LIN {X 0,Y 162.743,Z 569.001,A -85,B 0,C 180,E1 -23228.066,E2 -23228.066} C_VEL
LIN {X 0,Y 163.505,Z 560.276,A -85,B 0,C 180,E1 -23232.409,E2 -23232.409} C_VEL
LIN {X 0,Y 164.914,Z 549.825,A -85,B 0,C 180,E1 -23236.716,E2 -23236.716} C_VEL
LIN {X 0,Y 166.509,Z 539.199,A -85,B 0,C 180,E1 -23240.376,E2 -23240.376} C_VEL
LIN {X 0,Y 168.483,Z 527.294,A -85,B 0,C 180,E1 -23243.803,E2 -23243.803} C_VEL
LIN {X 0,Y 170.774,Z 514.351,A -85,B 0,C 180,E1 -23246.914,E2 -23246.914} C_VEL
LIN {X 0,Y 173.276,Z 499.762,A -85,B 0,C 180,E1 -23249.79,E2 -23249.79} C_VEL
LIN {X 0,Y 175.692,Z 484.547,A -85,B 0,C 180,E1 -23252.203,E2 -23252.203} C_VEL
LIN {X 0,Y 177.954,Z 468.333,A -85,B 0,C 180,E1 -23254.246,E2 -23254.246} C_VEL
LIN {X 0,Y 179.877,Z 451.506,A -85,B 0,C 180,E1 -23255.876,E2 -23255.876} C_VEL
LIN {X 0,Y 183.136,Z 416.504,A -85,B 0,C 180,E1 -23258.314,E2 -23258.314} C_VEL
LIN {X 0,Y 188.818,Z 360.63,A -85,B 0,C 180,E1 -23261.887,E2 -23261.887} C_VEL
LIN {X 0,Y 177.895,Z 334.141,A -85,B 0,C 180,E1 -23265.296,E2 -23265.296} C_VEL
LIN {X 0,Y 167.703,Z 310.796,A -85,B 0,C 180,E1 -23268.793,E2 -23268.793} C_VEL
LIN {X 0,Y 164.401,Z 303.304,A -85,B 0,C 180,E1 -23270.012,E2 -23270.012} C_VEL
LIN {X 0,Y 164.284,Z 302.644,A -85,B 0,C 180,E1 -23270.145,E2 -23270.145} C_VEL
LIN {X 0,Y 164.33,Z 302.638,A -85,B 0,C 180,E1 -23274.345,E2 -23274.345} C_VEL
LIN {X 0,Y 164.369,Z 302.631,A -85,B 0,C 180,E1 -23279.127,E2 -23279.127} C_VEL
LIN {X 0,Y 164.392,Z 302.632,A -85,B 0,C 180,E1 -23284.687,E2 -23284.687} C_VEL
LIN {X 0,Y 164.435,Z 302.629,A -85,B 0,C 180,E1 -23290.092,E2 -23290.092} C_VEL
LIN {X 0,Y 164.485,Z 302.624,A -85,B 0,C 180,E1 -23295.142,E2 -23295.142} C_VEL
LIN {X 0,Y 164.797,Z 302.585,A -85,B 0,C 180,E1 -23300.175,E2 -23300.175} C_VEL
LIN {X 0,Y 164.846,Z 302.576,A -85,B 0,C 180,E1 -23302.648,E2 -23302.648} C_VEL
LIN {X 0,Y 165.043,Z 302.554,A -85,B 0,C 180,E1 -23307.556,E2 -23307.556} C_VEL
LIN {X 0,Y 165.289,Z 302.518,A -85,B 0,C 180,E1 -23309.997,E2 -23309.997} C_VEL
LIN {X 0,Y 164.765,Z 302.585,A -85,B 0,C 180,E1 -23314.89,E2 -23314.89} C_VEL
LIN {X 0,Y 164.847,Z 302.577,A -85,B 0,C 180,E1 -23317.345,E2 -23317.345} C_VEL
LIN {X 0,Y 164.735,Z 302.585,A -85,B 0,C 180,E1 -23321.129,E2 -23321.129} C_VEL
LIN {X 0,Y 164.475,Z 302.619,A -85,B 0,C 180,E1 -23327.4,E2 -23327.4} C_VEL
LIN {X 0,Y 164.464,Z 302.621,A -85,B 0,C 180,E1 -23329.987,E2 -23329.987} C_VEL
LIN {X 0,Y 164.383,Z 302.629,A -85,B 0,C 180,E1 -23336.131,E2 -23336.131} C_VEL
LIN {X 0,Y 164.363,Z 302.637,A -85,B 0,C 180,E1 -23341.225,E2 -23341.225} C_VEL
LIN {X 0,Y 164.3,Z 302.64,A -85,B 0,C 180,E1 -23346.783,E2 -23346.783} C_VEL
LIN {X 0,Y 164.288,Z 302.645,A -85,B 0,C 180,E1 -23349.912,E2 -23349.912} C_VEL
LIN {X 0,Y 164.267,Z 302.644,A -85,B 0,C 180,E1 -23353.341,E2 -23353.341} C_VEL
LIN {X 0,Y 164.251,Z 302.649,A -85,B 0,C 180,E1 -23356.798,E2 -23356.798} C_VEL
LIN {X 0,Y 164.283,Z 302.644,A -85,B 0,C 180,E1 -23360.351,E2 -23360.351} C_VEL
LIN {X 0,Y 164.317,Z 302.641,A -85,B 0,C 180,E1 -23366.222,E2 -23366.222} C_VEL
LIN {X 0,Y 164.393,Z 302.63,A -85,B 0,C 180,E1 -23369.138,E2 -23369.138} C_VEL
LIN {X 0,Y 164.394,Z 302.632,A -85,B 0,C 180,E1 -23374.693,E2 -23374.693} C_VEL
LIN {X 0,Y 164.472,Z 302.618,A -85,B 0,C 180,E1 -23380.052,E2 -23380.052} C_VEL
LIN {X 0,Y 164.524,Z 302.616,A -85,B 0,C 180,E1 -23385.151,E2 -23385.151} C_VEL
LIN {X 0,Y 164.797,Z 302.58,A -85,B 0,C 180,E1 -23390.18,E2 -23390.18} C_VEL
LIN {X 0,Y 164.839,Z 302.577,A -85,B 0,C 180,E1 -23392.653,E2 -23392.653} C_VEL
LIN {X 0,Y 165.038,Z 302.551,A -85,B 0,C 180,E1 -23397.561,E2 -23397.561} C_VEL
LIN {X 0,Y 165.285,Z 302.52,A -85,B 0,C 180,E1 -23400.002,E2 -23400.002} C_VEL
LIN {X 0,Y 164.76,Z 302.587,A -85,B 0,C 180,E1 -23404.896,E2 -23404.896} C_VEL
LIN {X 0,Y 164.841,Z 302.576,A -85,B 0,C 180,E1 -23407.35,E2 -23407.35} C_VEL
LIN {X 0,Y 164.745,Z 302.59,A -85,B 0,C 180,E1 -23411.154,E2 -23411.154} C_VEL
LIN {X 0,Y 164.476,Z 302.624,A -85,B 0,C 180,E1 -23417.406,E2 -23417.406} C_VEL
LIN {X 0,Y 164.465,Z 302.626,A -85,B 0,C 180,E1 -23419.992,E2 -23419.992} C_VEL
LIN {X 0,Y 164.379,Z 302.637,A -85,B 0,C 180,E1 -23426.131,E2 -23426.131} C_VEL
LIN {X 0,Y 164.382,Z 302.636,A -85,B 0,C 180,E1 -23431.239,E2 -23431.239} C_VEL
LIN {X 0,Y 164.351,Z 302.637,A -85,B 0,C 180,E1 -23437.545,E2 -23437.545} C_VEL
LIN {X 0,Y 164.407,Z 302.858,A -85,B 0,C 180,E1 -23438.014,E2 -23438.014} C_VEL
LIN {X 0,Y 174.424,Z 329.86,A -85,B 0,C 180,E1 -23441.961,E2 -23441.961} C_VEL
LIN {X 0,Y 184.34,Z 358.027,A -85,B 0,C 180,E1 -23445.535,E2 -23445.535} C_VEL
LIN {X 0,Y 188.983,Z 371.855,A -85,B 0,C 180,E1 -23447.122,E2 -23447.122} C_VEL
LIN {X 0,Y 189.295,Z 378.263,A -85,B 0,C 180,E1 -23447.63,E2 -23447.63} C_VEL
LIN {X 0,Y 180.179,Z 471.457,A -85,B 0,C 180,E1 -23453.85,E2 -23453.85} C_VEL
LIN {X 0,Y 178.064,Z 488.079,A -85,B 0,C 180,E1 -23455.437,E2 -23455.437} C_VEL
LIN {X 0,Y 175.518,Z 504.903,A -85,B 0,C 180,E1 -23457.572,E2 -23457.572} C_VEL
LIN {X 0,Y 172.894,Z 520.655,A -85,B 0,C 180,E1 -23460.139,E2 -23460.139} C_VEL
LIN {X 0,Y 170.429,Z 534.802,A -85,B 0,C 180,E1 -23463.029,E2 -23463.029} C_VEL
LIN {X 0,Y 168.143,Z 547.791,A -85,B 0,C 180,E1 -23466.283,E2 -23466.283} C_VEL
LIN {X 0,Y 167.894,Z 549.217,A -85,B 0,C 180,E1 -23466.688,E2 -23466.688} C_VEL
LIN {X 0,Y 166.516,Z 553.567,A -85,B 0,C 180,E1 -23467.983,E2 -23467.983} C_VEL
LIN {X 0,Y 162.593,Z 560.027,A -85,B 0,C 180,E1 -23470.217,E2 -23470.217} C_VEL
LIN {X 0,Y 158.866,Z 566.141,A -85,B 0,C 180,E1 -23472.686,E2 -23472.686} C_VEL
LIN {X 0,Y 157.82,Z 569.902,A -85,B 0,C 180,E1 -23474.303,E2 -23474.303} C_VEL
LIN {X 0,Y 157.069,Z 578.706,A -85,B 0,C 180,E1 -23478.388,E2 -23478.388} C_VEL
LIN {X 0,Y 156.845,Z 586.764,A -85,B 0,C 180,E1 -23482.925,E2 -23482.925} C_VEL
LIN {X 0,Y 156.901,Z 591.497,A -85,B 0,C 180,E1 -23486.151,E2 -23486.151} C_VEL
LIN {X 0,Y 156.999,Z 596.192,A -85,B 0,C 180,E1 -23490.004,E2 -23490.004} C_VEL
LIN {X 0,Y 156.404,Z 599.726,A -85,B 0,C 180,E1 -23493.868,E2 -23493.868} C_VEL
LIN {X 0,Y 156.018,Z 602.437,A -85,B 0,C 180,E1 -23497.77,E2 -23497.77} C_VEL
LIN {X 0,Y 156.148,Z 605.076,A -85,B 0,C 180,E1 -23503.009,E2 -23503.009} C_VEL
LIN {X 0,Y 157.589,Z 606.716,A -85,B 0,C 180,E1 -23508.194,E2 -23508.194} C_VEL
LIN {X 0,Y 160.486,Z 607.537,A -85,B 0,C 180,E1 -23513.215,E2 -23513.215} C_VEL
LIN {X 0,Y 167.481,Z 607.223,A -85,B 0,C 180,E1 -23520.239,E2 -23520.239} C_VEL
LIN {X 0,Y 177.074,Z 605.132,A -85,B 0,C 180,E1 -23526.541,E2 -23526.541} C_VEL
LIN {X 0,Y 185.072,Z 602.786,A -85,B 0,C 180,E1 -23530.211,E2 -23530.211} C_VEL
LIN {X 0,Y 194.013,Z 599.774,A -85,B 0,C 180,E1 -23533.496,E2 -23533.496} C_VEL
LIN {X 0,Y 205.058,Z 595.453,A -85,B 0,C 180,E1 -23536.726,E2 -23536.726} C_VEL
LIN {X 0,Y 205.719,Z 595.098,A -85,B 0,C 180,E1 -23537.233,E2 -23537.233} C_VEL
LIN {X 0,Y 196.732,Z 597.398,A -85,B 0,C 180,E1 -23539.98,E2 -23539.98} C_VEL
LIN {X 0,Y 183.81,Z 599.568,A -85,B 0,C 180,E1 -23545.002,E2 -23545.002} C_VEL
LIN {X 0,Y 176.253,Z 599.98,A -85,B 0,C 180,E1 -23548.775,E2 -23548.775} C_VEL
LIN {X 0,Y 169.945,Z 599.539,A -85,B 0,C 180,E1 -23552.94,E2 -23552.94} C_VEL
LIN {X 0,Y 164.67,Z 598.231,A -85,B 0,C 180,E1 -23557.409,E2 -23557.409} C_VEL
LIN {X 0,Y 160.779,Z 596.017,A -85,B 0,C 180,E1 -23562.181,E2 -23562.181} C_VEL
LIN {X 0,Y 157.895,Z 592.902,A -85,B 0,C 180,E1 -23567.139,E2 -23567.139} C_VEL
LIN {X 0,Y 155.901,Z 587.493,A -85,B 0,C 180,E1 -23573.533,E2 -23573.533} C_VEL
LIN {X 0,Y 155.54,Z 583.386,A -85,B 0,C 180,E1 -23577.408,E2 -23577.408} C_VEL
LIN {X 0,Y 155.366,Z 578.521,A -85,B 0,C 180,E1 -23581.294,E2 -23581.294} C_VEL
LIN {X 0,Y 155.54,Z 571.047,A -85,B 0,C 180,E1 -23586.222,E2 -23586.222} C_VEL
LIN {X 0,Y 156.083,Z 563.476,A -85,B 0,C 180,E1 -23590.374,E2 -23590.374} C_VEL
LIN {X 0,Y 157.215,Z 553.624,A -85,B 0,C 180,E1 -23594.892,E2 -23594.892} C_VEL
LIN {X 0,Y 158.614,Z 543.638,A -85,B 0,C 180,E1 -23598.736,E2 -23598.736} C_VEL
LIN {X 0,Y 160.777,Z 530.826,A -85,B 0,C 180,E1 -23602.825,E2 -23602.825} C_VEL
LIN {X 0,Y 163.25,Z 516.685,A -85,B 0,C 180,E1 -23606.527,E2 -23606.527} C_VEL
LIN {X 0,Y 165.685,Z 502.525,A -85,B 0,C 180,E1 -23609.543,E2 -23609.543} C_VEL
LIN {X 0,Y 168.246,Z 487.239,A -85,B 0,C 180,E1 -23612.178,E2 -23612.178} C_VEL
LIN {X 0,Y 170.757,Z 470.23,A -85,B 0,C 180,E1 -23614.477,E2 -23614.477} C_VEL
LIN {X 0,Y 172.789,Z 453.3,A -85,B 0,C 180,E1 -23616.228,E2 -23616.228} C_VEL
LIN {X 0,Y 175.716,Z 422.77,A -85,B 0,C 180,E1 -23618.492,E2 -23618.492} C_VEL
LIN {X 0,Y 181.978,Z 362.013,A -85,B 0,C 180,E1 -23622.588,E2 -23622.588} C_VEL
LIN {X 0,Y 171.144,Z 335.711,A -85,B 0,C 180,E1 -23626.13,E2 -23626.13} C_VEL
LIN {X 0,Y 160.884,Z 312.149,A -85,B 0,C 180,E1 -23629.833,E2 -23629.833} C_VEL
LIN {X 0,Y 157.365,Z 304.37,A -85,B 0,C 180,E1 -23631.187,E2 -23631.187} C_VEL
LIN {X 0,Y 157.203,Z 303.526,A -85,B 0,C 180,E1 -23631.408,E2 -23631.408} C_VEL
LIN {X 0,Y 157.278,Z 303.516,A -85,B 0,C 180,E1 -23634.482,E2 -23634.482} C_VEL
LIN {X 0,Y 157.282,Z 303.516,A -85,B 0,C 180,E1 -23638.098,E2 -23638.098} C_VEL
LIN {X 0,Y 157.307,Z 303.515,A -85,B 0,C 180,E1 -23643.46,E2 -23643.46} C_VEL
LIN {X 0,Y 157.374,Z 303.511,A -85,B 0,C 180,E1 -23649.681,E2 -23649.681} C_VEL
LIN {X 0,Y 157.419,Z 303.504,A -85,B 0,C 180,E1 -23654.459,E2 -23654.459} C_VEL
LIN {X 0,Y 157.722,Z 303.468,A -85,B 0,C 180,E1 -23659.729,E2 -23659.729} C_VEL
LIN {X 0,Y 157.803,Z 303.453,A -85,B 0,C 180,E1 -23662.318,E2 -23662.318} C_VEL
LIN {X 0,Y 158.251,Z 303.395,A -85,B 0,C 180,E1 -23669.997,E2 -23669.997} C_VEL
LIN {X 0,Y 157.803,Z 303.452,A -85,B 0,C 180,E1 -23677.675,E2 -23677.675} C_VEL
LIN {X 0,Y 157.665,Z 303.466,A -85,B 0,C 180,E1 -23681.299,E2 -23681.299} C_VEL
LIN {X 0,Y 157.446,Z 303.498,A -85,B 0,C 180,E1 -23685.531,E2 -23685.531} C_VEL
LIN {X 0,Y 157.361,Z 303.506,A -85,B 0,C 180,E1 -23690.93,E2 -23690.93} C_VEL
LIN {X 0,Y 157.304,Z 303.51,A -85,B 0,C 180,E1 -23696.682,E2 -23696.682} C_VEL
LIN {X 0,Y 157.265,Z 303.519,A -85,B 0,C 180,E1 -23702.425,E2 -23702.425} C_VEL
LIN {X 0,Y 157.269,Z 303.515,A -85,B 0,C 180,E1 -23706.454,E2 -23706.454} C_VEL
LIN {X 0,Y 157.201,Z 303.525,A -85,B 0,C 180,E1 -23712.109,E2 -23712.109} C_VEL
LIN {X 0,Y 157.181,Z 303.53,A -85,B 0,C 180,E1 -23717.883,E2 -23717.883} C_VEL
LIN {X 0,Y 157.255,Z 303.519,A -85,B 0,C 180,E1 -23723.55,E2 -23723.55} C_VEL
LIN {X 0,Y 157.289,Z 303.515,A -85,B 0,C 180,E1 -23728.091,E2 -23728.091} C_VEL
LIN {X 0,Y 157.303,Z 303.516,A -85,B 0,C 180,E1 -23733.465,E2 -23733.465} C_VEL
LIN {X 0,Y 157.38,Z 303.502,A -85,B 0,C 180,E1 -23739.67,E2 -23739.67} C_VEL
LIN {X 0,Y 157.45,Z 303.496,A -85,B 0,C 180,E1 -23744.468,E2 -23744.468} C_VEL
LIN {X 0,Y 157.723,Z 303.461,A -85,B 0,C 180,E1 -23749.735,E2 -23749.735} C_VEL
LIN {X 0,Y 157.797,Z 303.453,A -85,B 0,C 180,E1 -23752.324,E2 -23752.324} C_VEL
LIN {X 0,Y 158.247,Z 303.396,A -85,B 0,C 180,E1 -23760.002,E2 -23760.002} C_VEL
LIN {X 0,Y 157.799,Z 303.453,A -85,B 0,C 180,E1 -23767.68,E2 -23767.68} C_VEL
LIN {X 0,Y 157.673,Z 303.47,A -85,B 0,C 180,E1 -23771.322,E2 -23771.322} C_VEL
LIN {X 0,Y 157.453,Z 303.498,A -85,B 0,C 180,E1 -23775.536,E2 -23775.536} C_VEL
LIN {X 0,Y 157.359,Z 303.513,A -85,B 0,C 180,E1 -23780.936,E2 -23780.936} C_VEL
LIN {X 0,Y 157.302,Z 303.52,A -85,B 0,C 180,E1 -23786.684,E2 -23786.684} C_VEL
LIN {X 0,Y 157.275,Z 303.521,A -85,B 0,C 180,E1 -23792.43,E2 -23792.43} C_VEL
LIN {X 0,Y 157.299,Z 303.662,A -85,B 0,C 180,E1 -23796.782,E2 -23796.782} C_VEL
LIN {X 0,Y 158.315,Z 306.417,A -85,B 0,C 180,E1 -23797.23,E2 -23797.23} C_VEL
LIN {X 0,Y 161.302,Z 313.749,A -85,B 0,C 180,E1 -23798.451,E2 -23798.451} C_VEL
LIN {X 0,Y 170.717,Z 339.571,A -85,B 0,C 180,E1 -23802.219,E2 -23802.219} C_VEL
LIN {X 0,Y 181.836,Z 371.924,A -85,B 0,C 180,E1 -23806.307,E2 -23806.307} C_VEL
LIN {X 0,Y 182.488,Z 374.64,A -85,B 0,C 180,E1 -23806.593,E2 -23806.593} C_VEL
LIN {X 0,Y 182.512,Z 379.17,A -85,B 0,C 180,E1 -23806.945,E2 -23806.945} C_VEL
LIN {X 0,Y 173.291,Z 470.889,A -85,B 0,C 180,E1 -23813.354,E2 -23813.354} C_VEL
LIN {X 0,Y 171.029,Z 488.174,A -85,B 0,C 180,E1 -23815.09,E2 -23815.09} C_VEL
LIN {X 0,Y 168.568,Z 504.001,A -85,B 0,C 180,E1 -23817.184,E2 -23817.184} C_VEL
LIN {X 0,Y 165.952,Z 519.55,A -85,B 0,C 180,E1 -23819.812,E2 -23819.812} C_VEL
LIN {X 0,Y 163.44,Z 533.752,A -85,B 0,C 180,E1 -23822.818,E2 -23822.818} C_VEL
LIN {X 0,Y 160.98,Z 547.649,A -85,B 0,C 180,E1 -23826.468,E2 -23826.468} C_VEL
LIN {X 0,Y 159.258,Z 558.77,A -85,B 0,C 180,E1 -23830.005,E2 -23830.005} C_VEL
LIN {X 0,Y 157.82,Z 569.902,A -85,B 0,C 180,E1 -23834.303,E2 -23834.303} C_VEL
LIN {X 0,Y 156.843,Z 573.57,A -85,B 0,C 180,E1 -23835.974,E2 -23835.974} C_VEL
LIN {X 0,Y 153.579,Z 578.678,A -85,B 0,C 180,E1 -23838.872,E2 -23838.872} C_VEL
LIN {X 0,Y 150.589,Z 583.4,A -85,B 0,C 180,E1 -23841.995,E2 -23841.995} C_VEL
LIN {X 0,Y 150.048,Z 586.324,A -85,B 0,C 180,E1 -23843.952,E2 -23843.952} C_VEL
LIN {X 0,Y 150.095,Z 592.612,A -85,B 0,C 180,E1 -23848.662,E2 -23848.662} C_VEL
LIN {X 0,Y 150.058,Z 595.5,A -85,B 0,C 180,E1 -23851.346,E2 -23851.346} C_VEL
LIN {X 0,Y 149.38,Z 598.925,A -85,B 0,C 180,E1 -23855.403,E2 -23855.403} C_VEL
LIN {X 0,Y 149.055,Z 602.289,A -85,B 0,C 180,E1 -23860.875,E2 -23860.875} C_VEL
LIN {X 0,Y 149.939,Z 604.692,A -85,B 0,C 180,E1 -23866.337,E2 -23866.337} C_VEL
LIN {X 0,Y 153.688,Z 606.534,A -85,B 0,C 180,E1 -23873.85,E2 -23873.85} C_VEL
LIN {X 0,Y 158.571,Z 606.846,A -85,B 0,C 180,E1 -23879.182,E2 -23879.182} C_VEL
LIN {X 0,Y 164.389,Z 606.36,A -85,B 0,C 180,E1 -23883.768,E2 -23883.768} C_VEL
LIN {X 0,Y 171.405,Z 605.089,A -85,B 0,C 180,E1 -23887.958,E2 -23887.958} C_VEL
LIN {X 0,Y 179.732,Z 603.155,A -85,B 0,C 180,E1 -23891.666,E2 -23891.666} C_VEL
LIN {X 0,Y 188.963,Z 600.49,A -85,B 0,C 180,E1 -23894.967,E2 -23894.967} C_VEL
LIN {X 0,Y 196.373,Z 598.06,A -85,B 0,C 180,E1 -23897.155,E2 -23897.155} C_VEL
LIN {X 0,Y 186.819,Z 599.715,A -85,B 0,C 180,E1 -23900.242,E2 -23900.242} C_VEL
LIN {X 0,Y 178.099,Z 600.588,A -85,B 0,C 180,E1 -23903.705,E2 -23903.705} C_VEL
LIN {X 0,Y 170.245,Z 600.644,A -85,B 0,C 180,E1 -23907.542,E2 -23907.542} C_VEL
LIN {X 0,Y 163.653,Z 599.866,A -85,B 0,C 180,E1 -23911.809,E2 -23911.809} C_VEL
LIN {X 0,Y 158.138,Z 598.221,A -85,B 0,C 180,E1 -23916.421,E2 -23916.421} C_VEL
LIN {X 0,Y 154.048,Z 595.742,A -85,B 0,C 180,E1 -23921.374,E2 -23921.374} C_VEL
LIN {X 0,Y 150.434,Z 591.275,A -85,B 0,C 180,E1 -23927.862,E2 -23927.862} C_VEL
LIN {X 0,Y 148.924,Z 586.344,A -85,B 0,C 180,E1 -23933.393,E2 -23933.393} C_VEL
LIN {X 0,Y 148.548,Z 582.223,A -85,B 0,C 180,E1 -23937.286,E2 -23937.286} C_VEL
LIN {X 0,Y 148.356,Z 577.075,A -85,B 0,C 180,E1 -23941.355,E2 -23941.355} C_VEL
LIN {X 0,Y 148.596,Z 569.035,A -85,B 0,C 180,E1 -23946.652,E2 -23946.652} C_VEL
LIN {X 0,Y 149.305,Z 559.986,A -85,B 0,C 180,E1 -23951.538,E2 -23951.538} C_VEL
LIN {X 0,Y 150.691,Z 549.471,A -85,B 0,C 180,E1 -23956.248,E2 -23956.248} C_VEL
LIN {X 0,Y 152.242,Z 538.695,A -85,B 0,C 180,E1 -23960.254,E2 -23960.254} C_VEL
LIN {X 0,Y 154.419,Z 526.049,A -85,B 0,C 180,E1 -23964.178,E2 -23964.178} C_VEL
LIN {X 0,Y 156.905,Z 512.255,A -85,B 0,C 180,E1 -23967.689,E2 -23967.689} C_VEL
LIN {X 0,Y 159.536,Z 497.226,A -85,B 0,C 180,E1 -23970.802,E2 -23970.802} C_VEL
LIN {X 0,Y 162.227,Z 480.769,A -85,B 0,C 180,E1 -23973.526,E2 -23973.526} C_VEL
LIN {X 0,Y 164.6,Z 463.974,A -85,B 0,C 180,E1 -23975.659,E2 -23975.659} C_VEL
LIN {X 0,Y 166.526,Z 446.338,A -85,B 0,C 180,E1 -23977.347,E2 -23977.347} C_VEL
LIN {X 0,Y 175.189,Z 363.631,A -85,B 0,C 180,E1 -23983.28,E2 -23983.28} C_VEL
LIN {X 0,Y 164.621,Z 337.772,A -85,B 0,C 180,E1 -23986.912,E2 -23986.912} C_VEL
LIN {X 0,Y 153.612,Z 312.55,A -85,B 0,C 180,E1 -23991.099,E2 -23991.099} C_VEL
LIN {X 0,Y 150.299,Z 305.128,A -85,B 0,C 180,E1 -23992.454,E2 -23992.454} C_VEL
LIN {X 0,Y 150.197,Z 304.402,A -85,B 0,C 180,E1 -23992.639,E2 -23992.639} C_VEL
LIN {X 0,Y 150.208,Z 304.402,A -85,B 0,C 180,E1 -23997.368,E2 -23997.368} C_VEL
LIN {X 0,Y 150.237,Z 304.395,A -85,B 0,C 180,E1 -24002.718,E2 -24002.718} C_VEL
LIN {X 0,Y 150.336,Z 304.386,A -85,B 0,C 180,E1 -24009.216,E2 -24009.216} C_VEL
LIN {X 0,Y 150.327,Z 304.389,A -85,B 0,C 180,E1 -24013.706,E2 -24013.706} C_VEL
LIN {X 0,Y 150.643,Z 304.347,A -85,B 0,C 180,E1 -24019.241,E2 -24019.241} C_VEL
LIN {X 0,Y 150.737,Z 304.335,A -85,B 0,C 180,E1 -24021.956,E2 -24021.956} C_VEL
LIN {X 0,Y 151.212,Z 304.272,A -85,B 0,C 180,E1 -24029.996,E2 -24029.996} C_VEL
LIN {X 0,Y 150.737,Z 304.331,A -85,B 0,C 180,E1 -24038.037,E2 -24038.037} C_VEL
LIN {X 0,Y 150.599,Z 304.347,A -85,B 0,C 180,E1 -24041.489,E2 -24041.489} C_VEL
LIN {X 0,Y 150.353,Z 304.379,A -85,B 0,C 180,E1 -24046.284,E2 -24046.284} C_VEL
LIN {X 0,Y 150.342,Z 304.38,A -85,B 0,C 180,E1 -24050.79,E2 -24050.79} C_VEL
LIN {X 0,Y 150.234,Z 304.391,A -85,B 0,C 180,E1 -24057.279,E2 -24057.279} C_VEL
LIN {X 0,Y 150.206,Z 304.398,A -85,B 0,C 180,E1 -24062.631,E2 -24062.631} C_VEL
LIN {X 0,Y 150.199,Z 304.399,A -85,B 0,C 180,E1 -24067.46,E2 -24067.46} C_VEL
LIN {X 0,Y 150.142,Z 304.406,A -85,B 0,C 180,E1 -24071.505,E2 -24071.505} C_VEL
LIN {X 0,Y 150.114,Z 304.408,A -85,B 0,C 180,E1 -24075.394,E2 -24075.394} C_VEL
LIN {X 0,Y 150.129,Z 304.41,A -85,B 0,C 180,E1 -24079.055,E2 -24079.055} C_VEL
LIN {X 0,Y 150.167,Z 304.398,A -85,B 0,C 180,E1 -24082.707,E2 -24082.707} C_VEL
LIN {X 0,Y 150.208,Z 304.399,A -85,B 0,C 180,E1 -24087.364,E2 -24087.364} C_VEL
LIN {X 0,Y 150.23,Z 304.394,A -85,B 0,C 180,E1 -24092.72,E2 -24092.72} C_VEL
LIN {X 0,Y 150.337,Z 304.378,A -85,B 0,C 180,E1 -24099.21,E2 -24099.21} C_VEL
LIN {X 0,Y 150.355,Z 304.38,A -85,B 0,C 180,E1 -24103.715,E2 -24103.715} C_VEL
LIN {X 0,Y 150.647,Z 304.342,A -85,B 0,C 180,E1 -24109.247,E2 -24109.247} C_VEL
LIN {X 0,Y 150.733,Z 304.333,A -85,B 0,C 180,E1 -24111.961,E2 -24111.961} C_VEL
LIN {X 0,Y 151.207,Z 304.273,A -85,B 0,C 180,E1 -24120.002,E2 -24120.002} C_VEL
LIN {X 0,Y 150.735,Z 304.333,A -85,B 0,C 180,E1 -24128.043,E2 -24128.043} C_VEL
LIN {X 0,Y 150.605,Z 304.35,A -85,B 0,C 180,E1 -24131.509,E2 -24131.509} C_VEL
LIN {X 0,Y 150.358,Z 304.381,A -85,B 0,C 180,E1 -24136.289,E2 -24136.289} C_VEL
LIN {X 0,Y 150.341,Z 304.388,A -85,B 0,C 180,E1 -24140.794,E2 -24140.794} C_VEL
LIN {X 0,Y 150.235,Z 304.4,A -85,B 0,C 180,E1 -24147.284,E2 -24147.284} C_VEL
LIN {X 0,Y 150.214,Z 304.401,A -85,B 0,C 180,E1 -24152.639,E2 -24152.639} C_VEL
LIN {X 0,Y 150.236,Z 304.456,A -85,B 0,C 180,E1 -24155.478,E2 -24155.478} C_VEL
LIN {X 0,Y 151.342,Z 307.401,A -85,B 0,C 180,E1 -24155.998,E2 -24155.998} C_VEL
LIN {X 0,Y 155.149,Z 316.348,A -85,B 0,C 180,E1 -24157.6,E2 -24157.6} C_VEL
LIN {X 0,Y 165.144,Z 344.15,A -85,B 0,C 180,E1 -24161.8,E2 -24161.8} C_VEL
LIN {X 0,Y 175.848,Z 375.839,A -85,B 0,C 180,E1 -24165.903,E2 -24165.903} C_VEL
LIN {X 0,Y 175.79,Z 379.632,A -85,B 0,C 180,E1 -24166.204,E2 -24166.204} C_VEL
LIN {X 0,Y 166.312,Z 470.815,A -85,B 0,C 180,E1 -24172.884,E2 -24172.884} C_VEL
LIN {X 0,Y 164.08,Z 487.65,A -85,B 0,C 180,E1 -24174.664,E2 -24174.664} C_VEL
LIN {X 0,Y 161.405,Z 504.564,A -85,B 0,C 180,E1 -24177.029,E2 -24177.029} C_VEL
LIN {X 0,Y 158.753,Z 519.866,A -85,B 0,C 180,E1 -24179.768,E2 -24179.768} C_VEL
LIN {X 0,Y 156.251,Z 533.879,A -85,B 0,C 180,E1 -24182.913,E2 -24182.913} C_VEL
LIN {X 0,Y 153.765,Z 547.716,A -85,B 0,C 180,E1 -24186.771,E2 -24186.771} C_VEL
LIN {X 0,Y 152.121,Z 558.605,A -85,B 0,C 180,E1 -24190.435,E2 -24190.435} C_VEL
LIN {X 0,Y 150.733,Z 570.096,A -85,B 0,C 180,E1 -24195.145,E2 -24195.145} C_VEL
LIN {X 0,Y 150.111,Z 579.525,A -85,B 0,C 180,E1 -24199.861,E2 -24199.861} C_VEL
LIN {X 0,Y 150.048,Z 586.324,A -85,B 0,C 180,E1 -24203.952,E2 -24203.952} C_VEL
LIN {X 0,Y 149.834,Z 588.215,A -85,B 0,C 180,E1 -24205.266,E2 -24205.266} C_VEL
LIN {X 0,Y 148.545,Z 590.565,A -85,B 0,C 180,E1 -24207.297,E2 -24207.297} C_VEL
LIN {X 0,Y 145.272,Z 593.542,A -85,B 0,C 180,E1 -24210.822,E2 -24210.822} C_VEL
LIN {X 0,Y 142.774,Z 596.194,A -85,B 0,C 180,E1 -24214.609,E2 -24214.609} C_VEL
LIN {X 0,Y 142.601,Z 596.764,A -85,B 0,C 180,E1 -24215.389,E2 -24215.389} C_VEL
LIN {X 0,Y 142.246,Z 600.628,A -85,B 0,C 180,E1 -24221.402,E2 -24221.402} C_VEL
LIN {X 0,Y 143.22,Z 603.202,A -85,B 0,C 180,E1 -24227.127,E2 -24227.127} C_VEL
LIN {X 0,Y 145.736,Z 604.978,A -85,B 0,C 180,E1 -24232.697,E2 -24232.697} C_VEL
LIN {X 0,Y 152.402,Z 606.079,A -85,B 0,C 180,E1 -24240.486,E2 -24240.486} C_VEL
LIN {X 0,Y 162.069,Z 605.502,A -85,B 0,C 180,E1 -24247.384,E2 -24247.384} C_VEL
LIN {X 0,Y 170.003,Z 604.221,A -85,B 0,C 180,E1 -24251.414,E2 -24251.414} C_VEL
LIN {X 0,Y 179.121,Z 602.303,A -85,B 0,C 180,E1 -24254.934,E2 -24254.934} C_VEL
LIN {X 0,Y 186.339,Z 600.452,A -85,B 0,C 180,E1 -24257.241,E2 -24257.241} C_VEL
LIN {X 0,Y 176.904,Z 601.31,A -85,B 0,C 180,E1 -24260.53,E2 -24260.53} C_VEL
LIN {X 0,Y 168.18,Z 601.442,A -85,B 0,C 180,E1 -24264.192,E2 -24264.192} C_VEL
LIN {X 0,Y 160.72,Z 600.704,A -85,B 0,C 180,E1 -24268.347,E2 -24268.347} C_VEL
LIN {X 0,Y 154.401,Z 599.185,A -85,B 0,C 180,E1 -24272.922,E2 -24272.922} C_VEL
LIN {X 0,Y 149.333,Z 596.791,A -85,B 0,C 180,E1 -24277.881,E2 -24277.881} C_VEL
LIN {X 0,Y 145.588,Z 593.528,A -85,B 0,C 180,E1 -24283.162,E2 -24283.162} C_VEL
LIN {X 0,Y 143.054,Z 589.303,A -85,B 0,C 180,E1 -24288.665,E2 -24288.665} C_VEL
LIN {X 0,Y 141.701,Z 582.493,A -85,B 0,C 180,E1 -24295.731,E2 -24295.731} C_VEL
LIN {X 0,Y 141.438,Z 577.375,A -85,B 0,C 180,E1 -24299.998,E2 -24299.998} C_VEL
LIN {X 0,Y 141.473,Z 570.237,A -85,B 0,C 180,E1 -24305.025,E2 -24305.025} C_VEL
LIN {X 0,Y 142.03,Z 561.784,A -85,B 0,C 180,E1 -24309.971,E2 -24309.971} C_VEL
LIN {X 0,Y 143.185,Z 551.587,A -85,B 0,C 180,E1 -24314.93,E2 -24314.93} C_VEL
LIN {X 0,Y 144.652,Z 541.167,A -85,B 0,C 180,E1 -24319.142,E2 -24319.142} C_VEL
LIN {X 0,Y 146.903,Z 528.042,A -85,B 0,C 180,E1 -24323.567,E2 -24323.567} C_VEL
LIN {X 0,Y 149.341,Z 514.703,A -85,B 0,C 180,E1 -24327.234,E2 -24327.234} C_VEL
LIN {X 0,Y 152.006,Z 499.843,A -85,B 0,C 180,E1 -24330.567,E2 -24330.567} C_VEL
LIN {X 0,Y 154.703,Z 483.909,A -85,B 0,C 180,E1 -24333.421,E2 -24333.421} C_VEL
LIN {X 0,Y 157.179,Z 467.239,A -85,B 0,C 180,E1 -24335.761,E2 -24335.761} C_VEL
LIN {X 0,Y 159.317,Z 449.832,A -85,B 0,C 180,E1 -24337.601,E2 -24337.601} C_VEL
LIN {X 0,Y 168.361,Z 365.029,A -85,B 0,C 180,E1 -24344.026,E2 -24344.026} C_VEL
LIN {X 0,Y 157.138,Z 337.641,A -85,B 0,C 180,E1 -24348.081,E2 -24348.081} C_VEL
LIN {X 0,Y 146.528,Z 313.374,A -85,B 0,C 180,E1 -24352.372,E2 -24352.372} C_VEL
LIN {X 0,Y 143.196,Z 305.821,A -85,B 0,C 180,E1 -24353.847,E2 -24353.847} C_VEL
LIN {X 0,Y 143.093,Z 305.283,A -85,B 0,C 180,E1 -24354.069,E2 -24354.069} C_VEL
LIN {X 0,Y 143.175,Z 305.278,A -85,B 0,C 180,E1 -24357.315,E2 -24357.315} C_VEL
LIN {X 0,Y 143.181,Z 305.275,A -85,B 0,C 180,E1 -24362.065,E2 -24362.065} C_VEL
LIN {X 0,Y 143.264,Z 305.266,A -85,B 0,C 180,E1 -24368.752,E2 -24368.752} C_VEL
LIN {X 0,Y 143.265,Z 305.266,A -85,B 0,C 180,E1 -24372.879,E2 -24372.879} C_VEL
LIN {X 0,Y 143.59,Z 305.225,A -85,B 0,C 180,E1 -24378.706,E2 -24378.706} C_VEL
LIN {X 0,Y 143.657,Z 305.219,A -85,B 0,C 180,E1 -24381.557,E2 -24381.557} C_VEL
LIN {X 0,Y 144.171,Z 305.149,A -85,B 0,C 180,E1 -24389.996,E2 -24389.996} C_VEL
LIN {X 0,Y 143.656,Z 305.212,A -85,B 0,C 180,E1 -24398.436,E2 -24398.436} C_VEL
LIN {X 0,Y 143.54,Z 305.228,A -85,B 0,C 180,E1 -24401.709,E2 -24401.709} C_VEL
LIN {X 0,Y 143.293,Z 305.259,A -85,B 0,C 180,E1 -24407.11,E2 -24407.11} C_VEL
LIN {X 0,Y 143.268,Z 305.263,A -85,B 0,C 180,E1 -24411.252,E2 -24411.252} C_VEL
LIN {X 0,Y 143.18,Z 305.272,A -85,B 0,C 180,E1 -24417.934,E2 -24417.934} C_VEL
LIN {X 0,Y 143.156,Z 305.276,A -85,B 0,C 180,E1 -24423.432,E2 -24423.432} C_VEL
LIN {X 0,Y 143.063,Z 305.289,A -85,B 0,C 180,E1 -24429.684,E2 -24429.684} C_VEL
LIN {X 0,Y 143.045,Z 305.286,A -85,B 0,C 180,E1 -24433.453,E2 -24433.453} C_VEL
LIN {X 0,Y 143.027,Z 305.295,A -85,B 0,C 180,E1 -24437.475,E2 -24437.475} C_VEL
LIN {X 0,Y 143.063,Z 305.283,A -85,B 0,C 180,E1 -24441.807,E2 -24441.807} C_VEL
LIN {X 0,Y 143.175,Z 305.276,A -85,B 0,C 180,E1 -24447.322,E2 -24447.322} C_VEL
LIN {X 0,Y 143.178,Z 305.271,A -85,B 0,C 180,E1 -24452.064,E2 -24452.064} C_VEL
LIN {X 0,Y 143.263,Z 305.26,A -85,B 0,C 180,E1 -24458.749,E2 -24458.749} C_VEL
LIN {X 0,Y 143.293,Z 305.261,A -85,B 0,C 180,E1 -24462.888,E2 -24462.888} C_VEL
LIN {X 0,Y 143.583,Z 305.219,A -85,B 0,C 180,E1 -24468.712,E2 -24468.712} C_VEL
LIN {X 0,Y 143.654,Z 305.216,A -85,B 0,C 180,E1 -24471.563,E2 -24471.563} C_VEL
LIN {X 0,Y 144.166,Z 305.15,A -85,B 0,C 180,E1 -24480.002,E2 -24480.002} C_VEL
LIN {X 0,Y 143.655,Z 305.215,A -85,B 0,C 180,E1 -24488.442,E2 -24488.442} C_VEL
LIN {X 0,Y 143.539,Z 305.23,A -85,B 0,C 180,E1 -24491.715,E2 -24491.715} C_VEL
LIN {X 0,Y 143.296,Z 305.264,A -85,B 0,C 180,E1 -24497.116,E2 -24497.116} C_VEL
LIN {X 0,Y 143.267,Z 305.268,A -85,B 0,C 180,E1 -24501.256,E2 -24501.256} C_VEL
LIN {X 0,Y 143.183,Z 305.278,A -85,B 0,C 180,E1 -24507.94,E2 -24507.94} C_VEL
LIN {X 0,Y 143.166,Z 305.277,A -85,B 0,C 180,E1 -24514.024,E2 -24514.024} C_VEL
LIN {X 0,Y 144.302,Z 308.361,A -85,B 0,C 180,E1 -24514.673,E2 -24514.673} C_VEL
LIN {X 0,Y 148.355,Z 317.459,A -85,B 0,C 180,E1 -24516.428,E2 -24516.428} C_VEL
LIN {X 0,Y 157.563,Z 342.945,A -85,B 0,C 180,E1 -24520.523,E2 -24520.523} C_VEL
LIN {X 0,Y 169.07,Z 376.982,A -85,B 0,C 180,E1 -24525.175,E2 -24525.175} C_VEL
LIN {X 0,Y 169.13,Z 379.479,A -85,B 0,C 180,E1 -24525.394,E2 -24525.394} C_VEL
LIN {X 0,Y 159.412,Z 470.244,A -85,B 0,C 180,E1 -24532.366,E2 -24532.366} C_VEL
LIN {X 0,Y 157.186,Z 486.509,A -85,B 0,C 180,E1 -24534.146,E2 -24534.146} C_VEL
LIN {X 0,Y 154.535,Z 503.007,A -85,B 0,C 180,E1 -24536.54,E2 -24536.54} C_VEL
LIN {X 0,Y 151.847,Z 518.413,A -85,B 0,C 180,E1 -24539.399,E2 -24539.399} C_VEL
LIN {X 0,Y 149.302,Z 532.58,A -85,B 0,C 180,E1 -24542.685,E2 -24542.685} C_VEL
LIN {X 0,Y 147.039,Z 545.173,A -85,B 0,C 180,E1 -24546.285,E2 -24546.285} C_VEL
LIN {X 0,Y 145.013,Z 558.331,A -85,B 0,C 180,E1 -24550.909,E2 -24550.909} C_VEL
LIN {X 0,Y 143.709,Z 569.736,A -85,B 0,C 180,E1 -24555.851,E2 -24555.851} C_VEL
LIN {X 0,Y 143.201,Z 578.959,A -85,B 0,C 180,E1 -24560.735,E2 -24560.735} C_VEL
LIN {X 0,Y 143.204,Z 584.751,A -85,B 0,C 180,E1 -24564.371,E2 -24564.371} C_VEL
LIN {X 0,Y 143.265,Z 590.313,A -85,B 0,C 180,E1 -24568.598,E2 -24568.598} C_VEL
LIN {X 0,Y 143.273,Z 593.4,A -85,B 0,C 180,E1 -24571.409,E2 -24571.409} C_VEL
LIN {X 0,Y 142.601,Z 596.764,A -85,B 0,C 180,E1 -24575.389,E2 -24575.389} C_VEL
LIN {X 0,Y 141.732,Z 598.21,A -85,B 0,C 180,E1 -24577.667,E2 -24577.667} C_VEL
LIN {X 0,Y 138.909,Z 599.63,A -85,B 0,C 180,E1 -24581.501,E2 -24581.501} C_VEL
LIN {X 0,Y 136.893,Z 600.514,A -85,B 0,C 180,E1 -24584.696,E2 -24584.696} C_VEL
LIN {X 0,Y 136.404,Z 601.314,A -85,B 0,C 180,E1 -24587.16,E2 -24587.16} C_VEL
LIN {X 0,Y 136.55,Z 601.641,A -85,B 0,C 180,E1 -24587.978,E2 -24587.978} C_VEL
LIN {X 0,Y 141.254,Z 604.324,A -85,B 0,C 180,E1 -24596.606,E2 -24596.606} C_VEL
LIN {X 0,Y 149.428,Z 605.284,A -85,B 0,C 180,E1 -24604.364,E2 -24604.364} C_VEL
LIN {X 0,Y 156.477,Z 605.008,A -85,B 0,C 180,E1 -24608.965,E2 -24608.965} C_VEL
LIN {X 0,Y 164.748,Z 604.104,A -85,B 0,C 180,E1 -24613.047,E2 -24613.047} C_VEL
LIN {X 0,Y 176.292,Z 602.08,A -85,B 0,C 180,E1 -24617.333,E2 -24617.333} C_VEL
LIN {X 0,Y 166.94,Z 602.227,A -85,B 0,C 180,E1 -24620.838,E2 -24620.838} C_VEL
LIN {X 0,Y 158.474,Z 601.533,A -85,B 0,C 180,E1 -24624.791,E2 -24624.791} C_VEL
LIN {X 0,Y 151.276,Z 600.107,A -85,B 0,C 180,E1 -24629.265,E2 -24629.265} C_VEL
LIN {X 0,Y 145.251,Z 597.796,A -85,B 0,C 180,E1 -24634.183,E2 -24634.183} C_VEL
LIN {X 0,Y 140.708,Z 594.717,A -85,B 0,C 180,E1 -24639.533,E2 -24639.533} C_VEL
LIN {X 0,Y 136.728,Z 589.508,A -85,B 0,C 180,E1 -24646.624,E2 -24646.624} C_VEL
LIN {X 0,Y 134.927,Z 582.66,A -85,B 0,C 180,E1 -24654.018,E2 -24654.018} C_VEL
LIN {X 0,Y 134.552,Z 577.583,A -85,B 0,C 180,E1 -24658.501,E2 -24658.501} C_VEL
LIN {X 0,Y 134.466,Z 570.556,A -85,B 0,C 180,E1 -24663.744,E2 -24663.744} C_VEL
LIN {X 0,Y 134.96,Z 562.115,A -85,B 0,C 180,E1 -24668.985,E2 -24668.985} C_VEL
LIN {X 0,Y 136.001,Z 551.966,A -85,B 0,C 180,E1 -24674.207,E2 -24674.207} C_VEL
LIN {X 0,Y 137.424,Z 541.63,A -85,B 0,C 180,E1 -24678.638,E2 -24678.638} C_VEL
LIN {X 0,Y 139.689,Z 528.434,A -85,B 0,C 180,E1 -24683.339,E2 -24683.339} C_VEL
LIN {X 0,Y 142.367,Z 513.739,A -85,B 0,C 180,E1 -24687.564,E2 -24687.564} C_VEL
LIN {X 0,Y 145.059,Z 499.033,A -85,B 0,C 180,E1 -24690.98,E2 -24690.98} C_VEL
LIN {X 0,Y 147.807,Z 482.918,A -85,B 0,C 180,E1 -24693.963,E2 -24693.963} C_VEL
LIN {X 0,Y 150.341,Z 466.222,A -85,B 0,C 180,E1 -24696.375,E2 -24696.375} C_VEL
LIN {X 0,Y 152.48,Z 448.675,A -85,B 0,C 180,E1 -24698.276,E2 -24698.276} C_VEL
LIN {X 0,Y 161.567,Z 366.699,A -85,B 0,C 180,E1 -24704.781,E2 -24704.781} C_VEL
LIN {X 0,Y 151.432,Z 341.663,A -85,B 0,C 180,E1 -24708.629,E2 -24708.629} C_VEL
LIN {X 0,Y 140.992,Z 317.47,A -85,B 0,C 180,E1 -24713.055,E2 -24713.055} C_VEL
LIN {X 0,Y 136.159,Z 306.684,A -85,B 0,C 180,E1 -24715.288,E2 -24715.288} C_VEL
LIN {X 0,Y 136.086,Z 306.158,A -85,B 0,C 180,E1 -24715.379,E2 -24715.379} C_VEL
LIN {X 0,Y 136.138,Z 306.152,A -85,B 0,C 180,E1 -24722.31,E2 -24722.31} C_VEL
LIN {X 0,Y 136.23,Z 306.143,A -85,B 0,C 180,E1 -24728.827,E2 -24728.827} C_VEL
LIN {X 0,Y 136.25,Z 306.142,A -85,B 0,C 180,E1 -24735.05,E2 -24735.05} C_VEL
LIN {X 0,Y 136.493,Z 306.109,A -85,B 0,C 180,E1 -24738.11,E2 -24738.11} C_VEL
LIN {X 0,Y 136.584,Z 306.1,A -85,B 0,C 180,E1 -24741.116,E2 -24741.116} C_VEL
LIN {X 0,Y 137.128,Z 306.026,A -85,B 0,C 180,E1 -24749.996,E2 -24749.996} C_VEL
LIN {X 0,Y 136.583,Z 306.094,A -85,B 0,C 180,E1 -24758.876,E2 -24758.876} C_VEL
LIN {X 0,Y 136.483,Z 306.108,A -85,B 0,C 180,E1 -24761.951,E2 -24761.951} C_VEL
LIN {X 0,Y 136.233,Z 306.133,A -85,B 0,C 180,E1 -24768.026,E2 -24768.026} C_VEL
LIN {X 0,Y 136.189,Z 306.146,A -85,B 0,C 180,E1 -24771.746,E2 -24771.746} C_VEL
LIN {X 0,Y 136.09,Z 306.154,A -85,B 0,C 180,E1 -24778.613,E2 -24778.613} C_VEL
LIN {X 0,Y 136.067,Z 306.157,A -85,B 0,C 180,E1 -24784.617,E2 -24784.617} C_VEL
LIN {X 0,Y 136.039,Z 306.165,A -85,B 0,C 180,E1 -24789.206,E2 -24789.206} C_VEL
LIN {X 0,Y 135.985,Z 306.165,A -85,B 0,C 180,E1 -24793.656,E2 -24793.656} C_VEL
LIN {X 0,Y 135.972,Z 306.172,A -85,B 0,C 180,E1 -24797.787,E2 -24797.787} C_VEL
LIN {X 0,Y 136.012,Z 306.161,A -85,B 0,C 180,E1 -24801.683,E2 -24801.683} C_VEL
LIN {X 0,Y 136.045,Z 306.163,A -85,B 0,C 180,E1 -24805.738,E2 -24805.738} C_VEL
LIN {X 0,Y 136.133,Z 306.149,A -85,B 0,C 180,E1 -24812.316,E2 -24812.316} C_VEL
LIN {X 0,Y 136.23,Z 306.135,A -85,B 0,C 180,E1 -24818.833,E2 -24818.833} C_VEL
LIN {X 0,Y 136.264,Z 306.136,A -85,B 0,C 180,E1 -24825.058,E2 -24825.058} C_VEL
LIN {X 0,Y 136.486,Z 306.102,A -85,B 0,C 180,E1 -24828.116,E2 -24828.116} C_VEL
LIN {X 0,Y 136.581,Z 306.098,A -85,B 0,C 180,E1 -24831.122,E2 -24831.122} C_VEL
LIN {X 0,Y 137.123,Z 306.028,A -85,B 0,C 180,E1 -24840.002,E2 -24840.002} C_VEL
LIN {X 0,Y 136.582,Z 306.098,A -85,B 0,C 180,E1 -24848.882,E2 -24848.882} C_VEL
LIN {X 0,Y 136.482,Z 306.109,A -85,B 0,C 180,E1 -24851.957,E2 -24851.957} C_VEL
LIN {X 0,Y 136.235,Z 306.142,A -85,B 0,C 180,E1 -24858.033,E2 -24858.033} C_VEL
LIN {X 0,Y 136.188,Z 306.149,A -85,B 0,C 180,E1 -24861.75,E2 -24861.75} C_VEL
LIN {X 0,Y 136.11,Z 306.16,A -85,B 0,C 180,E1 -24868.632,E2 -24868.632} C_VEL
LIN {X 0,Y 136.148,Z 306.153,A -85,B 0,C 180,E1 -24872.604,E2 -24872.604} C_VEL
LIN {X 0,Y 137.224,Z 309.144,A -85,B 0,C 180,E1 -24873.214,E2 -24873.214} C_VEL
LIN {X 0,Y 142.362,Z 320.573,A -85,B 0,C 180,E1 -24875.566,E2 -24875.566} C_VEL
LIN {X 0,Y 151.306,Z 345.604,A -85,B 0,C 180,E1 -24879.763,E2 -24879.763} C_VEL
LIN {X 0,Y 162.453,Z 378.874,A -85,B 0,C 180,E1 -24884.509,E2 -24884.509} C_VEL
LIN {X 0,Y 156.881,Z 428.184,A -85,B 0,C 180,E1 -24888.325,E2 -24888.325} C_VEL
LIN {X 0,Y 152.21,Z 471.455,A -85,B 0,C 180,E1 -24892.017,E2 -24892.017} C_VEL
LIN {X 0,Y 149.799,Z 488.828,A -85,B 0,C 180,E1 -24894.099,E2 -24894.099} C_VEL
LIN {X 0,Y 147.104,Z 505.144,A -85,B 0,C 180,E1 -24896.678,E2 -24896.678} C_VEL
LIN {X 0,Y 144.393,Z 519.944,A -85,B 0,C 180,E1 -24899.675,E2 -24899.675} C_VEL
LIN {X 0,Y 141.657,Z 534.864,A -85,B 0,C 180,E1 -24903.484,E2 -24903.484} C_VEL
LIN {X 0,Y 139.316,Z 548.375,A -85,B 0,C 180,E1 -24907.773,E2 -24907.773} C_VEL
LIN {X 0,Y 137.64,Z 559.668,A -85,B 0,C 180,E1 -24912.164,E2 -24912.164} C_VEL
LIN {X 0,Y 136.733,Z 569.293,A -85,B 0,C 180,E1 -24916.632,E2 -24916.632} C_VEL
LIN {X 0,Y 136.314,Z 578.554,A -85,B 0,C 180,E1 -24921.853,E2 -24921.853} C_VEL
LIN {X 0,Y 136.385,Z 584.122,A -85,B 0,C 180,E1 -24925.571,E2 -24925.571} C_VEL
LIN {X 0,Y 136.556,Z 589.608,A -85,B 0,C 180,E1 -24930.004,E2 -24930.004} C_VEL
LIN {X 0,Y 136.28,Z 592.533,A -85,B 0,C 180,E1 -24932.96,E2 -24932.96} C_VEL
LIN {X 0,Y 135.533,Z 597.003,A -85,B 0,C 180,E1 -24938.953,E2 -24938.953} C_VEL
LIN {X 0,Y 135.861,Z 600.322,A -85,B 0,C 180,E1 -24944.994,E2 -24944.994} C_VEL
LIN {X 0,Y 136.55,Z 601.641,A -85,B 0,C 180,E1 -24947.978,E2 -24947.978} C_VEL
LIN {X 0,Y 136.781,Z 602.483,A -85,B 0,C 180,E1 -24950.428,E2 -24950.428} C_VEL
LIN {X 0,Y 136.139,Z 603.121,A -85,B 0,C 180,E1 -24954.575,E2 -24954.575} C_VEL
LIN {X 0,Y 136.138,Z 603.34,A -85,B 0,C 180,E1 -24957.915,E2 -24957.915} C_VEL
LIN {X 0,Y 137.242,Z 603.564,A -85,B 0,C 180,E1 -24960.345,E2 -24960.345} C_VEL
LIN {X 0,Y 137.919,Z 603.677,A -85,B 0,C 180,E1 -24961.114,E2 -24961.114} C_VEL
LIN {X 0,Y 147.127,Z 604.455,A -85,B 0,C 180,E1 -24968.392,E2 -24968.392} C_VEL
LIN {X 0,Y 155.144,Z 604.163,A -85,B 0,C 180,E1 -24972.809,E2 -24972.809} C_VEL
LIN {X 0,Y 164.432,Z 603.275,A -85,B 0,C 180,E1 -24976.606,E2 -24976.606} C_VEL
LIN {X 0,Y 166.264,Z 603.019,A -85,B 0,C 180,E1 -24977.441,E2 -24977.441} C_VEL
LIN {X 0,Y 156.926,Z 602.353,A -85,B 0,C 180,E1 -24981.169,E2 -24981.169} C_VEL
LIN {X 0,Y 148.821,Z 600.971,A -85,B 0,C 180,E1 -24985.478,E2 -24985.478} C_VEL
LIN {X 0,Y 138.908,Z 597.379,A -85,B 0,C 180,E1 -24992.91,E2 -24992.91} C_VEL
LIN {X 0,Y 133.082,Z 592.977,A -85,B 0,C 180,E1 -24999.922,E2 -24999.922} C_VEL
LIN {X 0,Y 129.368,Z 587.08,A -85,B 0,C 180,E1 -25007.447,E2 -25007.447} C_VEL
LIN {X 0,Y 127.872,Z 579.498,A -85,B 0,C 180,E1 -25015.269,E2 -25015.269} C_VEL
LIN {X 0,Y 127.533,Z 572.846,A -85,B 0,C 180,E1 -25020.787,E2 -25020.787} C_VEL
LIN {X 0,Y 127.721,Z 564.848,A -85,B 0,C 180,E1 -25026.316,E2 -25026.316} C_VEL
LIN {X 0,Y 128.299,Z 556.757,A -85,B 0,C 180,E1 -25031.051,E2 -25031.051} C_VEL
LIN {X 0,Y 129.747,Z 545.59,A -85,B 0,C 180,E1 -25036.519,E2 -25036.519} C_VEL
LIN {X 0,Y 131.62,Z 533.074,A -85,B 0,C 180,E1 -25041.534,E2 -25041.534} C_VEL
LIN {X 0,Y 134.033,Z 519.933,A -85,B 0,C 180,E1 -25045.865,E2 -25045.865} C_VEL
LIN {X 0,Y 136.531,Z 506.19,A -85,B 0,C 180,E1 -25049.569,E2 -25049.569} C_VEL
LIN {X 0,Y 139.323,Z 491.185,A -85,B 0,C 180,E1 -25052.835,E2 -25052.835} C_VEL
LIN {X 0,Y 142.138,Z 474.357,A -85,B 0,C 180,E1 -25055.734,E2 -25055.734} C_VEL
LIN {X 0,Y 144.459,Z 457.897,A -85,B 0,C 180,E1 -25057.891,E2 -25057.891} C_VEL
LIN {X 0,Y 146.991,Z 435.619,A -85,B 0,C 180,E1 -25060.022,E2 -25060.022} C_VEL
LIN {X 0,Y 154.759,Z 368.192,A -85,B 0,C 180,E1 -25065.574,E2 -25065.574} C_VEL
LIN {X 0,Y 143.972,Z 341.535,A -85,B 0,C 180,E1 -25069.926,E2 -25069.926} C_VEL
LIN {X 0,Y 134.195,Z 318.767,A -85,B 0,C 180,E1 -25074.36,E2 -25074.36} C_VEL
LIN {X 0,Y 129.065,Z 307.56,A -85,B 0,C 180,E1 -25076.877,E2 -25076.877} C_VEL
LIN {X 0,Y 128.989,Z 307.045,A -85,B 0,C 180,E1 -25076.981,E2 -25076.981} C_VEL
LIN {X 0,Y 129.016,Z 307.038,A -85,B 0,C 180,E1 -25080.637,E2 -25080.637} C_VEL
LIN {X 0,Y 129.104,Z 307.028,A -85,B 0,C 180,E1 -25087.596,E2 -25087.596} C_VEL
LIN {X 0,Y 129.166,Z 307.025,A -85,B 0,C 180,E1 -25094.209,E2 -25094.209} C_VEL
LIN {X 0,Y 129.412,Z 306.991,A -85,B 0,C 180,E1 -25097.816,E2 -25097.816} C_VEL
LIN {X 0,Y 129.511,Z 306.981,A -85,B 0,C 180,E1 -25100.627,E2 -25100.627} C_VEL
LIN {X 0,Y 130.083,Z 306.903,A -85,B 0,C 180,E1 -25109.996,E2 -25109.996} C_VEL
LIN {X 0,Y 129.509,Z 306.973,A -85,B 0,C 180,E1 -25119.365,E2 -25119.365} C_VEL
LIN {X 0,Y 129.385,Z 306.991,A -85,B 0,C 180,E1 -25122.545,E2 -25122.545} C_VEL
LIN {X 0,Y 129.144,Z 307.016,A -85,B 0,C 180,E1 -25129.053,E2 -25129.053} C_VEL
LIN {X 0,Y 129.099,Z 307.028,A -85,B 0,C 180,E1 -25132.395,E2 -25132.395} C_VEL
LIN {X 0,Y 129.02,Z 307.034,A -85,B 0,C 180,E1 -25135.83,E2 -25135.83} C_VEL
LIN {X 0,Y 129.006,Z 307.039,A -85,B 0,C 180,E1 -25139.355,E2 -25139.355} C_VEL
LIN {X 0,Y 128.98,Z 307.038,A -85,B 0,C 180,E1 -25145.186,E2 -25145.186} C_VEL
LIN {X 0,Y 128.939,Z 307.049,A -85,B 0,C 180,E1 -25150.844,E2 -25150.844} C_VEL
LIN {X 0,Y 128.904,Z 307.048,A -85,B 0,C 180,E1 -25155.129,E2 -25155.129} C_VEL
LIN {X 0,Y 128.923,Z 307.049,A -85,B 0,C 180,E1 -25159.738,E2 -25159.738} C_VEL
LIN {X 0,Y 128.947,Z 307.046,A -85,B 0,C 180,E1 -25164.831,E2 -25164.831} C_VEL
LIN {X 0,Y 129.039,Z 307.03,A -85,B 0,C 180,E1 -25170.651,E2 -25170.651} C_VEL
LIN {X 0,Y 129.095,Z 307.025,A -85,B 0,C 180,E1 -25177.729,E2 -25177.729} C_VEL
LIN {X 0,Y 129.142,Z 307.02,A -85,B 0,C 180,E1 -25180.945,E2 -25180.945} C_VEL
LIN {X 0,Y 129.405,Z 306.984,A -85,B 0,C 180,E1 -25187.822,E2 -25187.822} C_VEL
LIN {X 0,Y 129.506,Z 306.977,A -85,B 0,C 180,E1 -25190.633,E2 -25190.633} C_VEL
LIN {X 0,Y 130.079,Z 306.905,A -85,B 0,C 180,E1 -25200.002,E2 -25200.002} C_VEL
LIN {X 0,Y 129.508,Z 306.977,A -85,B 0,C 180,E1 -25209.372,E2 -25209.372} C_VEL
LIN {X 0,Y 129.384,Z 306.994,A -85,B 0,C 180,E1 -25212.551,E2 -25212.551} C_VEL
LIN {X 0,Y 129.145,Z 307.027,A -85,B 0,C 180,E1 -25219.06,E2 -25219.06} C_VEL
LIN {X 0,Y 129.1,Z 307.033,A -85,B 0,C 180,E1 -25222.402,E2 -25222.402} C_VEL
LIN {X 0,Y 129.049,Z 307.038,A -85,B 0,C 180,E1 -25229.393,E2 -25229.393} C_VEL
LIN {X 0,Y 129.016,Z 307.042,A -85,B 0,C 180,E1 -25230.985,E2 -25230.985} C_VEL
LIN {X 0,Y 130.181,Z 310.083,A -85,B 0,C 180,E1 -25231.672,E2 -25231.672} C_VEL
LIN {X 0,Y 136.368,Z 323.663,A -85,B 0,C 180,E1 -25234.663,E2 -25234.663} C_VEL
LIN {X 0,Y 144.213,Z 345.87,A -85,B 0,C 180,E1 -25238.584,E2 -25238.584} C_VEL
LIN {X 0,Y 154.693,Z 377.443,A -85,B 0,C 180,E1 -25243.35,E2 -25243.35} C_VEL
LIN {X 0,Y 155.61,Z 380.891,A -85,B 0,C 180,E1 -25243.799,E2 -25243.799} C_VEL
LIN {X 0,Y 145.513,Z 469.558,A -85,B 0,C 180,E1 -25251.334,E2 -25251.334} C_VEL
LIN {X 0,Y 143.056,Z 486.7,A -85,B 0,C 180,E1 -25253.445,E2 -25253.445} C_VEL
LIN {X 0,Y 140.282,Z 503.21,A -85,B 0,C 180,E1 -25256.132,E2 -25256.132} C_VEL
LIN {X 0,Y 137.533,Z 518.263,A -85,B 0,C 180,E1 -25259.274,E2 -25259.274} C_VEL
LIN {X 0,Y 134.927,Z 532.368,A -85,B 0,C 180,E1 -25262.975,E2 -25262.975} C_VEL
LIN {X 0,Y 132.52,Z 545.901,A -85,B 0,C 180,E1 -25267.392,E2 -25267.392} C_VEL
LIN {X 0,Y 130.82,Z 557.461,A -85,B 0,C 180,E1 -25272.011,E2 -25272.011} C_VEL
LIN {X 0,Y 129.846,Z 567.774,A -85,B 0,C 180,E1 -25276.981,E2 -25276.981} C_VEL
LIN {X 0,Y 129.5,Z 576.744,A -85,B 0,C 180,E1 -25282.207,E2 -25282.207} C_VEL
LIN {X 0,Y 129.643,Z 583.398,A -85,B 0,C 180,E1 -25286.897,E2 -25286.897} C_VEL
LIN {X 0,Y 129.801,Z 588.779,A -85,B 0,C 180,E1 -25291.556,E2 -25291.556} C_VEL
LIN {X 0,Y 129.082,Z 592.727,A -85,B 0,C 180,E1 -25296.256,E2 -25296.256} C_VEL
LIN {X 0,Y 128.791,Z 596.846,A -85,B 0,C 180,E1 -25302.612,E2 -25302.612} C_VEL
LIN {X 0,Y 131.214,Z 601.125,A -85,B 0,C 180,E1 -25312.024,E2 -25312.024} C_VEL
LIN {X 0,Y 135.028,Z 602.954,A -85,B 0,C 180,E1 -25317.937,E2 -25317.937} C_VEL
LIN {X 0,Y 137.919,Z 603.677,A -85,B 0,C 180,E1 -25321.114,E2 -25321.114} C_VEL
LIN {X 0,Y 139.722,Z 603.942,A -85,B 0,C 180,E1 -25323.432,E2 -25323.432} C_VEL
LIN {X 0,Y 143.574,Z 603.748,A -85,B 0,C 180,E1 -25330.48,E2 -25330.48} C_VEL
LIN {X 0,Y 146.058,Z 603.622,A -85,B 0,C 180,E1 -25332.595,E2 -25332.595} C_VEL
LIN {X 0,Y 147.164,Z 603.591,A -85,B 0,C 180,E1 -25333.229,E2 -25333.229} C_VEL
LIN {X 0,Y 154.7,Z 603.326,A -85,B 0,C 180,E1 -25336.63,E2 -25336.63} C_VEL
LIN {X 0,Y 156.22,Z 603.157,A -85,B 0,C 180,E1 -25337.558,E2 -25337.558} C_VEL
LIN {X 0,Y 147.129,Z 601.803,A -85,B 0,C 180,E1 -25341.61,E2 -25341.61} C_VEL
LIN {X 0,Y 135.785,Z 598.34,A -85,B 0,C 180,E1 -25348.827,E2 -25348.827} C_VEL
LIN {X 0,Y 129.928,Z 594.989,A -85,B 0,C 180,E1 -25354.356,E2 -25354.356} C_VEL
LIN {X 0,Y 124.678,Z 589.637,A -85,B 0,C 180,E1 -25361.936,E2 -25361.936} C_VEL
LIN {X 0,Y 121.632,Z 582.71,A -85,B 0,C 180,E1 -25370.015,E2 -25370.015} C_VEL
LIN {X 0,Y 121.002,Z 577.73,A -85,B 0,C 180,E1 -25374.999,E2 -25374.999} C_VEL
LIN {X 0,Y 120.641,Z 570.771,A -85,B 0,C 180,E1 -25380.832,E2 -25380.832} C_VEL
LIN {X 0,Y 120.849,Z 562.435,A -85,B 0,C 180,E1 -25386.677,E2 -25386.677} C_VEL
LIN {X 0,Y 121.647,Z 552.375,A -85,B 0,C 180,E1 -25392.51,E2 -25392.51} C_VEL
LIN {X 0,Y 123.044,Z 542.217,A -85,B 0,C 180,E1 -25397.447,E2 -25397.447} C_VEL
LIN {X 0,Y 125.165,Z 529.11,A -85,B 0,C 180,E1 -25402.705,E2 -25402.705} C_VEL
LIN {X 0,Y 127.75,Z 515.257,A -85,B 0,C 180,E1 -25407.218,E2 -25407.218} C_VEL
LIN {X 0,Y 130.583,Z 500.079,A -85,B 0,C 180,E1 -25411.195,E2 -25411.195} C_VEL
LIN {X 0,Y 133.445,Z 484.34,A -85,B 0,C 180,E1 -25414.48,E2 -25414.48} C_VEL
LIN {X 0,Y 136.109,Z 468.122,A -85,B 0,C 180,E1 -25417.117,E2 -25417.117} C_VEL
LIN {X 0,Y 138.419,Z 450.483,A -85,B 0,C 180,E1 -25419.274,E2 -25419.274} C_VEL
LIN {X 0,Y 147.876,Z 369.575,A -85,B 0,C 180,E1 -25426.426,E2 -25426.426} C_VEL
LIN {X 0,Y 137.936,Z 344.855,A -85,B 0,C 180,E1 -25430.653,E2 -25430.653} C_VEL
LIN {X 0,Y 128.853,Z 323.364,A -85,B 0,C 180,E1 -25435.017,E2 -25435.017} C_VEL
LIN {X 0,Y 122.885,Z 310.745,A -85,B 0,C 180,E1 -25438.056,E2 -25438.056} C_VEL
LIN {X 0,Y 121.905,Z 307.92,A -85,B 0,C 180,E1 -25438.739,E2 -25438.739} C_VEL
LIN {X 0,Y 121.937,Z 307.921,A -85,B 0,C 180,E1 -25442.538,E2 -25442.538} C_VEL
LIN {X 0,Y 122.024,Z 307.909,A -85,B 0,C 180,E1 -25447.142,E2 -25447.142} C_VEL
LIN {X 0,Y 122.079,Z 307.906,A -85,B 0,C 180,E1 -25453.266,E2 -25453.266} C_VEL
LIN {X 0,Y 122.327,Z 307.873,A -85,B 0,C 180,E1 -25457.592,E2 -25457.592} C_VEL
LIN {X 0,Y 122.441,Z 307.862,A -85,B 0,C 180,E1 -25460.08,E2 -25460.08} C_VEL
LIN {X 0,Y 122.599,Z 307.839,A -85,B 0,C 180,E1 -25466.709,E2 -25466.709} C_VEL
LIN {X 0,Y 123.037,Z 307.781,A -85,B 0,C 180,E1 -25469.996,E2 -25469.996} C_VEL
LIN {X 0,Y 122.44,Z 307.858,A -85,B 0,C 180,E1 -25476.587,E2 -25476.587} C_VEL
LIN {X 0,Y 122.439,Z 307.852,A -85,B 0,C 180,E1 -25479.911,E2 -25479.911} C_VEL
LIN {X 0,Y 122.253,Z 307.881,A -85,B 0,C 180,E1 -25483.289,E2 -25483.289} C_VEL
LIN {X 0,Y 122.036,Z 307.906,A -85,B 0,C 180,E1 -25490.21,E2 -25490.21} C_VEL
LIN {X 0,Y 121.974,Z 307.916,A -85,B 0,C 180,E1 -25493.781,E2 -25493.781} C_VEL
LIN {X 0,Y 121.919,Z 307.922,A -85,B 0,C 180,E1 -25500.161,E2 -25500.161} C_VEL
LIN {X 0,Y 121.9,Z 307.92,A -85,B 0,C 180,E1 -25506.187,E2 -25506.187} C_VEL
LIN {X 0,Y 121.872,Z 307.927,A -85,B 0,C 180,E1 -25511.443,E2 -25511.443} C_VEL
LIN {X 0,Y 121.852,Z 307.931,A -85,B 0,C 180,E1 -25518.565,E2 -25518.565} C_VEL
LIN {X 0,Y 121.899,Z 307.923,A -85,B 0,C 180,E1 -25524.796,E2 -25524.796} C_VEL
LIN {X 0,Y 121.928,Z 307.916,A -85,B 0,C 180,E1 -25529.828,E2 -25529.828} C_VEL
LIN {X 0,Y 121.97,Z 307.916,A -85,B 0,C 180,E1 -25536.216,E2 -25536.216} C_VEL
LIN {X 0,Y 122.033,Z 307.904,A -85,B 0,C 180,E1 -25539.788,E2 -25539.788} C_VEL
LIN {X 0,Y 122.352,Z 307.862,A -85,B 0,C 180,E1 -25547.528,E2 -25547.528} C_VEL
LIN {X 0,Y 122.436,Z 307.857,A -85,B 0,C 180,E1 -25550.087,E2 -25550.087} C_VEL
LIN {X 0,Y 122.595,Z 307.839,A -85,B 0,C 180,E1 -25556.716,E2 -25556.716} C_VEL
LIN {X 0,Y 123.032,Z 307.783,A -85,B 0,C 180,E1 -25560.003,E2 -25560.003} C_VEL
LIN {X 0,Y 122.436,Z 307.857,A -85,B 0,C 180,E1 -25566.595,E2 -25566.595} C_VEL
LIN {X 0,Y 122.438,Z 307.857,A -85,B 0,C 180,E1 -25569.918,E2 -25569.918} C_VEL
LIN {X 0,Y 122.253,Z 307.882,A -85,B 0,C 180,E1 -25573.297,E2 -25573.297} C_VEL
LIN {X 0,Y 122.037,Z 307.912,A -85,B 0,C 180,E1 -25580.217,E2 -25580.217} C_VEL
LIN {X 0,Y 121.975,Z 307.92,A -85,B 0,C 180,E1 -25583.789,E2 -25583.789} C_VEL
LIN {X 0,Y 122.019,Z 307.914,A -85,B 0,C 180,E1 -25589.28,E2 -25589.28} C_VEL
LIN {X 0,Y 123.034,Z 310.84,A -85,B 0,C 180,E1 -25589.955,E2 -25589.955} C_VEL
LIN {X 0,Y 130.194,Z 326.134,A -85,B 0,C 180,E1 -25593.597,E2 -25593.597} C_VEL
LIN {X 0,Y 139.354,Z 352.611,A -85,B 0,C 180,E1 -25598.443,E2 -25598.443} C_VEL
LIN {X 0,Y 148.798,Z 381.473,A -85,B 0,C 180,E1 -25602.92,E2 -25602.92} C_VEL
LIN {X 0,Y 141.352,Z 443.311,A -85,B 0,C 180,E1 -25608.29,E2 -25608.29} C_VEL
LIN {X 0,Y 138.253,Z 471.23,A -85,B 0,C 180,E1 -25611.024,E2 -25611.024} C_VEL
LIN {X 0,Y 135.798,Z 487.82,A -85,B 0,C 180,E1 -25613.25,E2 -25613.25} C_VEL
LIN {X 0,Y 132.878,Z 504.888,A -85,B 0,C 180,E1 -25616.27,E2 -25616.27} C_VEL
LIN {X 0,Y 130.086,Z 519.576,A -85,B 0,C 180,E1 -25619.623,E2 -25619.623} C_VEL
LIN {X 0,Y 127.563,Z 533.072,A -85,B 0,C 180,E1 -25623.476,E2 -25623.476} C_VEL
LIN {X 0,Y 125.29,Z 546.425,A -85,B 0,C 180,E1 -25628.189,E2 -25628.189} C_VEL
LIN {X 0,Y 123.773,Z 556.883,A -85,B 0,C 180,E1 -25632.661,E2 -25632.661} C_VEL
LIN {X 0,Y 122.944,Z 566.983,A -85,B 0,C 180,E1 -25637.83,E2 -25637.83} C_VEL
LIN {X 0,Y 122.733,Z 576.044,A -85,B 0,C 180,E1 -25643.428,E2 -25643.428} C_VEL
LIN {X 0,Y 122.925,Z 581.58,A -85,B 0,C 180,E1 -25647.547,E2 -25647.547} C_VEL
LIN {X 0,Y 123.126,Z 586.234,A -85,B 0,C 180,E1 -25651.64,E2 -25651.64} C_VEL
LIN {X 0,Y 122.669,Z 589.132,A -85,B 0,C 180,E1 -25654.934,E2 -25654.934} C_VEL
LIN {X 0,Y 122.081,Z 593.908,A -85,B 0,C 180,E1 -25661.848,E2 -25661.848} C_VEL
LIN {X 0,Y 123.469,Z 598.029,A -85,B 0,C 180,E1 -25669.974,E2 -25669.974} C_VEL
LIN {X 0,Y 128.525,Z 601.337,A -85,B 0,C 180,E1 -25678.962,E2 -25678.962} C_VEL
LIN {X 0,Y 137.968,Z 603.269,A -85,B 0,C 180,E1 -25687.686,E2 -25687.686} C_VEL
LIN {X 0,Y 147.164,Z 603.591,A -85,B 0,C 180,E1 -25693.229,E2 -25693.229} C_VEL
LIN {X 0,Y 148.228,Z 603.468,A -85,B 0,C 180,E1 -25694.339,E2 -25694.339} C_VEL
LIN {X 0,Y 148.103,Z 603.226,A -85,B 0,C 180,E1 -25695.556,E2 -25695.556} C_VEL
LIN {X 0,Y 146.55,Z 602.744,A -85,B 0,C 180,E1 -25697.314,E2 -25697.314} C_VEL
LIN {X 0,Y 143.177,Z 601.958,A -85,B 0,C 180,E1 -25699.37,E2 -25699.37} C_VEL
LIN {X 0,Y 133.273,Z 599.157,A -85,B 0,C 180,E1 -25704.687,E2 -25704.687} C_VEL
LIN {X 0,Y 123.612,Z 594.079,A -85,B 0,C 180,E1 -25712.943,E2 -25712.943} C_VEL
LIN {X 0,Y 118.069,Z 588.366,A -85,B 0,C 180,E1 -25720.887,E2 -25720.887} C_VEL
LIN {X 0,Y 114.844,Z 581.06,A -85,B 0,C 180,E1 -25729.418,E2 -25729.418} C_VEL
LIN {X 0,Y 114.172,Z 575.798,A -85,B 0,C 180,E1 -25734.699,E2 -25734.699} C_VEL
LIN {X 0,Y 113.787,Z 568.539,A -85,B 0,C 180,E1 -25740.882,E2 -25740.882} C_VEL
LIN {X 0,Y 114.07,Z 559.776,A -85,B 0,C 180,E1 -25747.075,E2 -25747.075} C_VEL
LIN {X 0,Y 114.952,Z 549.246,A -85,B 0,C 180,E1 -25753.251,E2 -25753.251} C_VEL
LIN {X 0,Y 116.41,Z 538.503,A -85,B 0,C 180,E1 -25758.476,E2 -25758.476} C_VEL
LIN {X 0,Y 118.558,Z 525.893,A -85,B 0,C 180,E1 -25763.583,E2 -25763.583} C_VEL
LIN {X 0,Y 121.341,Z 511.313,A -85,B 0,C 180,E1 -25768.369,E2 -25768.369} C_VEL
LIN {X 0,Y 124.195,Z 496.233,A -85,B 0,C 180,E1 -25772.324,E2 -25772.324} C_VEL
LIN {X 0,Y 127.158,Z 479.683,A -85,B 0,C 180,E1 -25775.714,E2 -25775.714} C_VEL
LIN {X 0,Y 129.739,Z 463.515,A -85,B 0,C 180,E1 -25778.281,E2 -25778.281} C_VEL
LIN {X 0,Y 131.915,Z 446.235,A -85,B 0,C 180,E1 -25780.361,E2 -25780.361} C_VEL
LIN {X 0,Y 141.112,Z 371.305,A -85,B 0,C 180,E1 -25787.272,E2 -25787.272} C_VEL
LIN {X 0,Y 132.001,Z 348.292,A -85,B 0,C 180,E1 -25791.391,E2 -25791.391} C_VEL
LIN {X 0,Y 122.938,Z 326.619,A -85,B 0,C 180,E1 -25795.997,E2 -25795.997} C_VEL
LIN {X 0,Y 117.013,Z 313.991,A -85,B 0,C 180,E1 -25799.226,E2 -25799.226} C_VEL
LIN {X 0,Y 114.97,Z 309.407,A -85,B 0,C 180,E1 -25800.449,E2 -25800.449} C_VEL
LIN {X 0,Y 114.879,Z 308.798,A -85,B 0,C 180,E1 -25800.693,E2 -25800.693} C_VEL
LIN {X 0,Y 114.943,Z 308.792,A -85,B 0,C 180,E1 -25806.505,E2 -25806.505} C_VEL
LIN {X 0,Y 114.985,Z 308.788,A -85,B 0,C 180,E1 -25812.201,E2 -25812.201} C_VEL
LIN {X 0,Y 115.26,Z 308.753,A -85,B 0,C 180,E1 -25817.304,E2 -25817.304} C_VEL
LIN {X 0,Y 115.382,Z 308.737,A -85,B 0,C 180,E1 -25822.998,E2 -25822.998} C_VEL
LIN {X 0,Y 115.989,Z 308.659,A -85,B 0,C 180,E1 -25829.995,E2 -25829.995} C_VEL
LIN {X 0,Y 115.382,Z 308.737,A -85,B 0,C 180,E1 -25836.992,E2 -25836.992} C_VEL
LIN {X 0,Y 115.276,Z 308.749,A -85,B 0,C 180,E1 -25842.733,E2 -25842.733} C_VEL
LIN {X 0,Y 115.003,Z 308.778,A -85,B 0,C 180,E1 -25847.786,E2 -25847.786} C_VEL
LIN {X 0,Y 114.938,Z 308.793,A -85,B 0,C 180,E1 -25853.49,E2 -25853.49} C_VEL
LIN {X 0,Y 114.853,Z 308.804,A -85,B 0,C 180,E1 -25861.061,E2 -25861.061} C_VEL
LIN {X 0,Y 114.791,Z 308.81,A -85,B 0,C 180,E1 -25867.745,E2 -25867.745} C_VEL
LIN {X 0,Y 114.781,Z 308.808,A -85,B 0,C 180,E1 -25872.718,E2 -25872.718} C_VEL
LIN {X 0,Y 114.776,Z 308.813,A -85,B 0,C 180,E1 -25877.662,E2 -25877.662} C_VEL
LIN {X 0,Y 114.773,Z 308.806,A -85,B 0,C 180,E1 -25882.745,E2 -25882.745} C_VEL
LIN {X 0,Y 114.85,Z 308.801,A -85,B 0,C 180,E1 -25888.938,E2 -25888.938} C_VEL
LIN {X 0,Y 114.934,Z 308.792,A -85,B 0,C 180,E1 -25896.51,E2 -25896.51} C_VEL
LIN {X 0,Y 115.001,Z 308.784,A -85,B 0,C 180,E1 -25902.211,E2 -25902.211} C_VEL
LIN {X 0,Y 115.273,Z 308.744,A -85,B 0,C 180,E1 -25907.264,E2 -25907.264} C_VEL
LIN {X 0,Y 115.377,Z 308.738,A -85,B 0,C 180,E1 -25913.005,E2 -25913.005} C_VEL
LIN {X 0,Y 115.985,Z 308.661,A -85,B 0,C 180,E1 -25920.003,E2 -25920.003} C_VEL
LIN {X 0,Y 115.378,Z 308.737,A -85,B 0,C 180,E1 -25927,E2 -25927} C_VEL
LIN {X 0,Y 115.276,Z 308.752,A -85,B 0,C 180,E1 -25932.741,E2 -25932.741} C_VEL
LIN {X 0,Y 115.005,Z 308.788,A -85,B 0,C 180,E1 -25937.794,E2 -25937.794} C_VEL
LIN {X 0,Y 114.95,Z 308.796,A -85,B 0,C 180,E1 -25943.509,E2 -25943.509} C_VEL
LIN {X 0,Y 114.941,Z 308.993,A -85,B 0,C 180,E1 -25947.422,E2 -25947.422} C_VEL
LIN {X 0,Y 116.014,Z 311.778,A -85,B 0,C 180,E1 -25948.127,E2 -25948.127} C_VEL
LIN {X 0,Y 122.932,Z 326.359,A -85,B 0,C 180,E1 -25951.913,E2 -25951.913} C_VEL
LIN {X 0,Y 125.953,Z 334.271,A -85,B 0,C 180,E1 -25953.619,E2 -25953.619} C_VEL
LIN {X 0,Y 134.424,Z 359.448,A -85,B 0,C 180,E1 -25958.321,E2 -25958.321} C_VEL
LIN {X 0,Y 142.018,Z 382.923,A -85,B 0,C 180,E1 -25962.104,E2 -25962.104} C_VEL
LIN {X 0,Y 131.676,Z 468.288,A -85,B 0,C 180,E1 -25970.178,E2 -25970.178} C_VEL
LIN {X 0,Y 129.123,Z 485.343,A -85,B 0,C 180,E1 -25972.494,E2 -25972.494} C_VEL
LIN {X 0,Y 126.122,Z 502.649,A -85,B 0,C 180,E1 -25975.659,E2 -25975.659} C_VEL
LIN {X 0,Y 123.3,Z 517.422,A -85,B 0,C 180,E1 -25979.142,E2 -25979.142} C_VEL
LIN {X 0,Y 120.737,Z 531.15,A -85,B 0,C 180,E1 -25983.19,E2 -25983.19} C_VEL
LIN {X 0,Y 118.375,Z 544.772,A -85,B 0,C 180,E1 -25988.224,E2 -25988.224} C_VEL
LIN {X 0,Y 116.761,Z 556.647,A -85,B 0,C 180,E1 -25993.62,E2 -25993.62} C_VEL
LIN {X 0,Y 116.088,Z 565.902,A -85,B 0,C 180,E1 -25998.658,E2 -25998.658} C_VEL
LIN {X 0,Y 116.069,Z 575.267,A -85,B 0,C 180,E1 -26004.794,E2 -26004.794} C_VEL
LIN {X 0,Y 116.381,Z 581.683,A -85,B 0,C 180,E1 -26010.005,E2 -26010.005} C_VEL
LIN {X 0,Y 116.35,Z 585.169,A -85,B 0,C 180,E1 -26013.468,E2 -26013.468} C_VEL
LIN {X 0,Y 115.511,Z 590.38,A -85,B 0,C 180,E1 -26020.522,E2 -26020.522} C_VEL
LIN {X 0,Y 116.123,Z 594.352,A -85,B 0,C 180,E1 -26027.619,E2 -26027.619} C_VEL
LIN {X 0,Y 118.514,Z 597.476,A -85,B 0,C 180,E1 -26034.531,E2 -26034.531} C_VEL
LIN {X 0,Y 125.712,Z 600.737,A -85,B 0,C 180,E1 -26043.995,E2 -26043.995} C_VEL
LIN {X 0,Y 136.357,Z 602.404,A -85,B 0,C 180,E1 -26052.075,E2 -26052.075} C_VEL
LIN {X 0,Y 145.078,Z 602.755,A -85,B 0,C 180,E1 -26056.611,E2 -26056.611} C_VEL
LIN {X 0,Y 146.162,Z 602.61,A -85,B 0,C 180,E1 -26057.685,E2 -26057.685} C_VEL
LIN {X 0,Y 133.42,Z 599.217,A -85,B 0,C 180,E1 -26064.587,E2 -26064.587} C_VEL
LIN {X 0,Y 133.273,Z 599.157,A -85,B 0,C 180,E1 -26064.687,E2 -26064.687} C_VEL
LIN {X 0,Y 129.78,Z 597.856,A -85,B 0,C 180,E1 -26066.668,E2 -26066.668} C_VEL
LIN {X 0,Y 123.028,Z 595.208,A -85,B 0,C 180,E1 -26069.713,E2 -26069.713} C_VEL
LIN {X 0,Y 117.878,Z 592.697,A -85,B 0,C 180,E1 -26072.338,E2 -26072.338} C_VEL
LIN {X 0,Y 114.877,Z 590.686,A -85,B 0,C 180,E1 -26074.657,E2 -26074.657} C_VEL
LIN {X 0,Y 114.15,Z 590.032,A -85,B 0,C 180,E1 -26075.518,E2 -26075.518} C_VEL
LIN {X 0,Y 109.877,Z 583.978,A -85,B 0,C 180,E1 -26083.271,E2 -26083.271} C_VEL
LIN {X 0,Y 107.577,Z 575.601,A -85,B 0,C 180,E1 -26092.489,E2 -26092.489} C_VEL
LIN {X 0,Y 107.035,Z 568.402,A -85,B 0,C 180,E1 -26099.057,E2 -26099.057} C_VEL
LIN {X 0,Y 107.104,Z 559.694,A -85,B 0,C 180,E1 -26105.646,E2 -26105.646} C_VEL
LIN {X 0,Y 107.762,Z 549.665,A -85,B 0,C 180,E1 -26111.945,E2 -26111.945} C_VEL
LIN {X 0,Y 109.251,Z 538.513,A -85,B 0,C 180,E1 -26117.789,E2 -26117.789} C_VEL
LIN {X 0,Y 111.556,Z 524.792,A -85,B 0,C 180,E1 -26123.676,E2 -26123.676} C_VEL
LIN {X 0,Y 114.228,Z 510.91,A -85,B 0,C 180,E1 -26128.475,E2 -26128.475} C_VEL
LIN {X 0,Y 117.147,Z 495.652,A -85,B 0,C 180,E1 -26132.676,E2 -26132.676} C_VEL
LIN {X 0,Y 120.237,Z 478.883,A -85,B 0,C 180,E1 -26136.282,E2 -26136.282} C_VEL
LIN {X 0,Y 122.867,Z 462.598,A -85,B 0,C 180,E1 -26138.988,E2 -26138.988} C_VEL
LIN {X 0,Y 125.011,Z 445.907,A -85,B 0,C 180,E1 -26141.072,E2 -26141.072} C_VEL
LIN {X 0,Y 134.217,Z 372.507,A -85,B 0,C 180,E1 -26148.254,E2 -26148.254} C_VEL
LIN {X 0,Y 124.234,Z 347.233,A -85,B 0,C 180,E1 -26153.098,E2 -26153.098} C_VEL
LIN {X 0,Y 115.845,Z 327.239,A -85,B 0,C 180,E1 -26157.718,E2 -26157.718} C_VEL
LIN {X 0,Y 109.247,Z 313.174,A -85,B 0,C 180,E1 -26161.672,E2 -26161.672} C_VEL
LIN {X 0,Y 107.946,Z 310.531,A -85,B 0,C 180,E1 -26162.488,E2 -26162.488} C_VEL
LIN {X 0,Y 107.76,Z 309.687,A -85,B 0,C 180,E1 -26162.831,E2 -26162.831} C_VEL
LIN {X 0,Y 107.905,Z 309.668,A -85,B 0,C 180,E1 -26166.991,E2 -26166.991} C_VEL
LIN {X 0,Y 108.019,Z 309.66,A -85,B 0,C 180,E1 -26174.91,E2 -26174.91} C_VEL
LIN {X 0,Y 108.271,Z 309.625,A -85,B 0,C 180,E1 -26178.766,E2 -26178.766} C_VEL
LIN {X 0,Y 108.451,Z 309.602,A -85,B 0,C 180,E1 -26186.279,E2 -26186.279} C_VEL
LIN {X 0,Y 108.939,Z 309.537,A -85,B 0,C 180,E1 -26189.995,E2 -26189.995} C_VEL
LIN {X 0,Y 108.321,Z 309.616,A -85,B 0,C 180,E1 -26197.451,E2 -26197.451} C_VEL
LIN {X 0,Y 108.191,Z 309.632,A -85,B 0,C 180,E1 -26203.011,E2 -26203.011} C_VEL
LIN {X 0,Y 107.896,Z 309.662,A -85,B 0,C 180,E1 -26209.001,E2 -26209.001} C_VEL
LIN {X 0,Y 107.848,Z 309.674,A -85,B 0,C 180,E1 -26214.18,E2 -26214.18} C_VEL
LIN {X 0,Y 107.78,Z 309.684,A -85,B 0,C 180,E1 -26222.045,E2 -26222.045} C_VEL
LIN {X 0,Y 107.696,Z 309.694,A -85,B 0,C 180,E1 -26228.461,E2 -26228.461} C_VEL
LIN {X 0,Y 107.663,Z 309.697,A -85,B 0,C 180,E1 -26235.886,E2 -26235.886} C_VEL
LIN {X 0,Y 107.673,Z 309.691,A -85,B 0,C 180,E1 -26241.551,E2 -26241.551} C_VEL
LIN {X 0,Y 107.785,Z 309.682,A -85,B 0,C 180,E1 -26248.562,E2 -26248.562} C_VEL
LIN {X 0,Y 107.898,Z 309.668,A -85,B 0,C 180,E1 -26256.998,E2 -26256.998} C_VEL
LIN {X 0,Y 108.026,Z 309.653,A -85,B 0,C 180,E1 -26264.919,E2 -26264.919} C_VEL
LIN {X 0,Y 108.277,Z 309.617,A -85,B 0,C 180,E1 -26268.775,E2 -26268.775} C_VEL
LIN {X 0,Y 108.446,Z 309.601,A -85,B 0,C 180,E1 -26276.287,E2 -26276.287} C_VEL
LIN {X 0,Y 108.935,Z 309.539,A -85,B 0,C 180,E1 -26280.003,E2 -26280.003} C_VEL
LIN {X 0,Y 108.319,Z 309.617,A -85,B 0,C 180,E1 -26287.459,E2 -26287.459} C_VEL
LIN {X 0,Y 108.19,Z 309.634,A -85,B 0,C 180,E1 -26293.02,E2 -26293.02} C_VEL
LIN {X 0,Y 107.896,Z 309.673,A -85,B 0,C 180,E1 -26299.01,E2 -26299.01} C_VEL
LIN {X 0,Y 107.849,Z 309.682,A -85,B 0,C 180,E1 -26305.015,E2 -26305.015} C_VEL
LIN {X 0,Y 107.835,Z 309.683,A -85,B 0,C 180,E1 -26305.246,E2 -26305.246} C_VEL
LIN {X 0,Y 108.858,Z 312.588,A -85,B 0,C 180,E1 -26306.041,E2 -26306.041} C_VEL
LIN {X 0,Y 113.045,Z 321.021,A -85,B 0,C 180,E1 -26308.566,E2 -26308.566} C_VEL
LIN {X 0,Y 118.703,Z 333.712,A -85,B 0,C 180,E1 -26311.827,E2 -26311.827} C_VEL
LIN {X 0,Y 127.063,Z 358.727,A -85,B 0,C 180,E1 -26316.857,E2 -26316.857} C_VEL
LIN {X 0,Y 135.232,Z 384.193,A -85,B 0,C 180,E1 -26321.225,E2 -26321.225} C_VEL
LIN {X 0,Y 124.698,Z 467.947,A -85,B 0,C 180,E1 -26329.605,E2 -26329.605} C_VEL
LIN {X 0,Y 122.105,Z 484.834,A -85,B 0,C 180,E1 -26332.044,E2 -26332.044} C_VEL
LIN {X 0,Y 119.088,Z 501.928,A -85,B 0,C 180,E1 -26335.346,E2 -26335.346} C_VEL
LIN {X 0,Y 116.124,Z 517.242,A -85,B 0,C 180,E1 -26339.202,E2 -26339.202} C_VEL
LIN {X 0,Y 113.413,Z 531.65,A -85,B 0,C 180,E1 -26343.805,E2 -26343.805} C_VEL
LIN {X 0,Y 111.349,Z 544.056,A -85,B 0,C 180,E1 -26348.726,E2 -26348.726} C_VEL
LIN {X 0,Y 109.867,Z 555.46,A -85,B 0,C 180,E1 -26354.249,E2 -26354.249} C_VEL
LIN {X 0,Y 109.297,Z 565.082,A -85,B 0,C 180,E1 -26359.82,E2 -26359.82} C_VEL
LIN {X 0,Y 109.462,Z 574.355,A -85,B 0,C 180,E1 -26366.324,E2 -26366.324} C_VEL
LIN {X 0,Y 109.838,Z 580.667,A -85,B 0,C 180,E1 -26371.838,E2 -26371.838} C_VEL
LIN {X 0,Y 109.799,Z 582.439,A -85,B 0,C 180,E1 -26373.675,E2 -26373.675} C_VEL
LIN {X 0,Y 109.102,Z 586.659,A -85,B 0,C 180,E1 -26379.272,E2 -26379.272} C_VEL
LIN {X 0,Y 109.68,Z 592.084,A -85,B 0,C 180,E1 -26388.691,E2 -26388.691} C_VEL
LIN {X 0,Y 114.431,Z 596.808,A -85,B 0,C 180,E1 -26399.433,E2 -26399.433} C_VEL
LIN {X 0,Y 123.428,Z 599.911,A -85,B 0,C 180,E1 -26408.786,E2 -26408.786} C_VEL
LIN {X 0,Y 135.648,Z 601.505,A -85,B 0,C 180,E1 -26416.503,E2 -26416.503} C_VEL
LIN {X 0,Y 136.557,Z 601.579,A -85,B 0,C 180,E1 -26416.947,E2 -26416.947} C_VEL
LIN {X 0,Y 136.321,Z 601.333,A -85,B 0,C 180,E1 -26417.914,E2 -26417.914} C_VEL
LIN {X 0,Y 127.442,Z 598.414,A -85,B 0,C 180,E1 -26422.939,E2 -26422.939} C_VEL
LIN {X 0,Y 118.894,Z 593.994,A -85,B 0,C 180,E1 -26429.835,E2 -26429.835} C_VEL
LIN {X 0,Y 114.15,Z 590.032,A -85,B 0,C 180,E1 -26435.518,E2 -26435.518} C_VEL
LIN {X 0,Y 111.789,Z 587.916,A -85,B 0,C 180,E1 -26438.043,E2 -26438.043} C_VEL
LIN {X 0,Y 106.867,Z 583.699,A -85,B 0,C 180,E1 -26441.976,E2 -26441.976} C_VEL
LIN {X 0,Y 102.563,Z 579.028,A -85,B 0,C 180,E1 -26446.17,E2 -26446.17} C_VEL
LIN {X 0,Y 101.284,Z 576.183,A -85,B 0,C 180,E1 -26449.021,E2 -26449.021} C_VEL
LIN {X 0,Y 100.447,Z 569.271,A -85,B 0,C 180,E1 -26455.985,E2 -26455.985} C_VEL
LIN {X 0,Y 100.19,Z 562.103,A -85,B 0,C 180,E1 -26462.007,E2 -26462.007} C_VEL
LIN {X 0,Y 100.441,Z 553.77,A -85,B 0,C 180,E1 -26468.041,E2 -26468.041} C_VEL
LIN {X 0,Y 101.616,Z 542.25,A -85,B 0,C 180,E1 -26474.976,E2 -26474.976} C_VEL
LIN {X 0,Y 103.354,Z 530.239,A -85,B 0,C 180,E1 -26480.912,E2 -26480.912} C_VEL
LIN {X 0,Y 105.712,Z 517.403,A -85,B 0,C 180,E1 -26486.129,E2 -26486.129} C_VEL
LIN {X 0,Y 108.141,Z 505.097,A -85,B 0,C 180,E1 -26490.239,E2 -26490.239} C_VEL
LIN {X 0,Y 111.338,Z 488.608,A -85,B 0,C 180,E1 -26494.614,E2 -26494.614} C_VEL
LIN {X 0,Y 114.265,Z 472.404,A -85,B 0,C 180,E1 -26497.952,E2 -26497.952} C_VEL
LIN {X 0,Y 116.95,Z 454.987,A -85,B 0,C 180,E1 -26500.662,E2 -26500.662} C_VEL
LIN {X 0,Y 122.419,Z 410.961,A -85,B 0,C 180,E1 -26505.56,E2 -26505.56} C_VEL
LIN {X 0,Y 127.407,Z 373.921,A -85,B 0,C 180,E1 -26509.234,E2 -26509.234} C_VEL
LIN {X 0,Y 117.731,Z 349.279,A -85,B 0,C 180,E1 -26514.273,E2 -26514.273} C_VEL
LIN {X 0,Y 109.864,Z 330.272,A -85,B 0,C 180,E1 -26518.946,E2 -26518.946} C_VEL
LIN {X 0,Y 103.678,Z 317.102,A -85,B 0,C 180,E1 -26522.901,E2 -26522.901} C_VEL
LIN {X 0,Y 100.962,Z 311.59,A -85,B 0,C 180,E1 -26524.757,E2 -26524.757} C_VEL
LIN {X 0,Y 100.786,Z 310.556,A -85,B 0,C 180,E1 -26525.02,E2 -26525.02} C_VEL
LIN {X 0,Y 100.802,Z 310.558,A -85,B 0,C 180,E1 -26529.592,E2 -26529.592} C_VEL
LIN {X 0,Y 101.169,Z 310.509,A -85,B 0,C 180,E1 -26537.966,E2 -26537.966} C_VEL
LIN {X 0,Y 101.258,Z 310.498,A -85,B 0,C 180,E1 -26542.015,E2 -26542.015} C_VEL
LIN {X 0,Y 101.863,Z 310.418,A -85,B 0,C 180,E1 -26549.995,E2 -26549.995} C_VEL
LIN {X 0,Y 101.26,Z 310.494,A -85,B 0,C 180,E1 -26557.973,E2 -26557.973} C_VEL
LIN {X 0,Y 101.117,Z 310.514,A -85,B 0,C 180,E1 -26563.347,E2 -26563.347} C_VEL
LIN {X 0,Y 100.808,Z 310.55,A -85,B 0,C 180,E1 -26570.395,E2 -26570.395} C_VEL
LIN {X 0,Y 100.765,Z 310.556,A -85,B 0,C 180,E1 -26574.955,E2 -26574.955} C_VEL
LIN {X 0,Y 100.687,Z 310.566,A -85,B 0,C 180,E1 -26583.119,E2 -26583.119} C_VEL
LIN {X 0,Y 100.642,Z 310.573,A -85,B 0,C 180,E1 -26589.818,E2 -26589.818} C_VEL
LIN {X 0,Y 100.634,Z 310.571,A -85,B 0,C 180,E1 -26595.709,E2 -26595.709} C_VEL
LIN {X 0,Y 100.611,Z 310.572,A -85,B 0,C 180,E1 -26601.052,E2 -26601.052} C_VEL
LIN {X 0,Y 100.679,Z 310.569,A -85,B 0,C 180,E1 -26606.884,E2 -26606.884} C_VEL
LIN {X 0,Y 100.775,Z 310.558,A -85,B 0,C 180,E1 -26615.268,E2 -26615.268} C_VEL
LIN {X 0,Y 100.804,Z 310.547,A -85,B 0,C 180,E1 -26619.602,E2 -26619.602} C_VEL
LIN {X 0,Y 101.177,Z 310.5,A -85,B 0,C 180,E1 -26627.975,E2 -26627.975} C_VEL
LIN {X 0,Y 101.256,Z 310.497,A -85,B 0,C 180,E1 -26632.024,E2 -26632.024} C_VEL
LIN {X 0,Y 101.859,Z 310.421,A -85,B 0,C 180,E1 -26640.003,E2 -26640.003} C_VEL
LIN {X 0,Y 101.258,Z 310.496,A -85,B 0,C 180,E1 -26647.982,E2 -26647.982} C_VEL
LIN {X 0,Y 101.116,Z 310.515,A -85,B 0,C 180,E1 -26653.356,E2 -26653.356} C_VEL
LIN {X 0,Y 100.88,Z 310.578,A -85,B 0,C 180,E1 -26662.939,E2 -26662.939} C_VEL
LIN {X 0,Y 101.866,Z 313.436,A -85,B 0,C 180,E1 -26663.78,E2 -26663.78} C_VEL
LIN {X 0,Y 107.669,Z 325.304,A -85,B 0,C 180,E1 -26667.582,E2 -26667.582} C_VEL
LIN {X 0,Y 112.844,Z 337.137,A -85,B 0,C 180,E1 -26670.791,E2 -26670.791} C_VEL
LIN {X 0,Y 120.737,Z 361.179,A -85,B 0,C 180,E1 -26675.889,E2 -26675.889} C_VEL
LIN {X 0,Y 128.39,Z 385.366,A -85,B 0,C 180,E1 -26680.272,E2 -26680.272} C_VEL
LIN {X 0,Y 117.639,Z 468.082,A -85,B 0,C 180,E1 -26689.065,E2 -26689.065} C_VEL
LIN {X 0,Y 114.949,Z 485.288,A -85,B 0,C 180,E1 -26691.76,E2 -26691.76} C_VEL
LIN {X 0,Y 112.02,Z 501.329,A -85,B 0,C 180,E1 -26695.088,E2 -26695.088} C_VEL
LIN {X 0,Y 109.147,Z 515.986,A -85,B 0,C 180,E1 -26699.001,E2 -26699.001} C_VEL
LIN {X 0,Y 106.603,Z 529.587,A -85,B 0,C 180,E1 -26703.582,E2 -26703.582} C_VEL
LIN {X 0,Y 104.34,Z 543.217,A -85,B 0,C 180,E1 -26709.297,E2 -26709.297} C_VEL
LIN {X 0,Y 102.974,Z 554.541,A -85,B 0,C 180,E1 -26715.176,E2 -26715.176} C_VEL
LIN {X 0,Y 102.546,Z 564.135,A -85,B 0,C 180,E1 -26721.135,E2 -26721.135} C_VEL
LIN {X 0,Y 102.852,Z 572.125,A -85,B 0,C 180,E1 -26727.068,E2 -26727.068} C_VEL
LIN {X 0,Y 103.225,Z 577.64,A -85,B 0,C 180,E1 -26731.956,E2 -26731.956} C_VEL
LIN {X 0,Y 103.29,Z 579.501,A -85,B 0,C 180,E1 -26733.907,E2 -26733.907} C_VEL
LIN {X 0,Y 102.643,Z 583.91,A -85,B 0,C 180,E1 -26739.862,E2 -26739.862} C_VEL
LIN {X 0,Y 103.368,Z 589.635,A -85,B 0,C 180,E1 -26749.879,E2 -26749.879} C_VEL
LIN {X 0,Y 106.288,Z 593.176,A -85,B 0,C 180,E1 -26757.577,E2 -26757.577} C_VEL
LIN {X 0,Y 111.925,Z 596.294,A -85,B 0,C 180,E1 -26765.28,E2 -26765.28} C_VEL
LIN {X 0,Y 122.046,Z 598.995,A -85,B 0,C 180,E1 -26773.716,E2 -26773.716} C_VEL
LIN {X 0,Y 127.258,Z 599.767,A -85,B 0,C 180,E1 -26776.841,E2 -26776.841} C_VEL
LIN {X 0,Y 126.503,Z 599.324,A -85,B 0,C 180,E1 -26778.187,E2 -26778.187} C_VEL
LIN {X 0,Y 116.344,Z 594.881,A -85,B 0,C 180,E1 -26784.977,E2 -26784.977} C_VEL
LIN {X 0,Y 108.585,Z 589.256,A -85,B 0,C 180,E1 -26793.057,E2 -26793.057} C_VEL
LIN {X 0,Y 103.263,Z 582.039,A -85,B 0,C 180,E1 -26802.347,E2 -26802.347} C_VEL
LIN {X 0,Y 101.284,Z 576.183,A -85,B 0,C 180,E1 -26809.021,E2 -26809.021} C_VEL
LIN {X 0,Y 100.216,Z 573.261,A -85,B 0,C 180,E1 -26811.851,E2 -26811.851} C_VEL
LIN {X 0,Y 98.41,Z 569.955,A -85,B 0,C 180,E1 -26814.49,E2 -26814.49} C_VEL
LIN {X 0,Y 94.544,Z 562.589,A -85,B 0,C 180,E1 -26819.693,E2 -26819.693} C_VEL
LIN {X 0,Y 93.527,Z 558.797,A -85,B 0,C 180,E1 -26822.473,E2 -26822.473} C_VEL
LIN {X 0,Y 93.466,Z 557.521,A -85,B 0,C 180,E1 -26823.435,E2 -26823.435} C_VEL
LIN {X 0,Y 93.814,Z 549.149,A -85,B 0,C 180,E1 -26829.447,E2 -26829.447} C_VEL
LIN {X 0,Y 95.076,Z 537.966,A -85,B 0,C 180,E1 -26836.215,E2 -26836.215} C_VEL
LIN {X 0,Y 97.191,Z 524.441,A -85,B 0,C 180,E1 -26842.868,E2 -26842.868} C_VEL
LIN {X 0,Y 99.873,Z 510.577,A -85,B 0,C 180,E1 -26848.355,E2 -26848.355} C_VEL
LIN {X 0,Y 102.873,Z 495.38,A -85,B 0,C 180,E1 -26853.126,E2 -26853.126} C_VEL
LIN {X 0,Y 105.702,Z 480.771,A -85,B 0,C 180,E1 -26856.751,E2 -26856.751} C_VEL
LIN {X 0,Y 108.644,Z 463.917,A -85,B 0,C 180,E1 -26859.97,E2 -26859.97} C_VEL
LIN {X 0,Y 111.15,Z 445.986,A -85,B 0,C 180,E1 -26862.51,E2 -26862.51} C_VEL
LIN {X 0,Y 120.627,Z 375.396,A -85,B 0,C 180,E1 -26870.272,E2 -26870.272} C_VEL
LIN {X 0,Y 111.503,Z 352.05,A -85,B 0,C 180,E1 -26875.353,E2 -26875.353} C_VEL
LIN {X 0,Y 104.195,Z 334.041,A -85,B 0,C 180,E1 -26880.032,E2 -26880.032} C_VEL
LIN {X 0,Y 98.193,Z 321.041,A -85,B 0,C 180,E1 -26884.194,E2 -26884.194} C_VEL
LIN {X 0,Y 94.985,Z 314.701,A -85,B 0,C 180,E1 -26886.56,E2 -26886.56} C_VEL
LIN {X 0,Y 93.777,Z 312.027,A -85,B 0,C 180,E1 -26887.552,E2 -26887.552} C_VEL
LIN {X 0,Y 93.699,Z 311.438,A -85,B 0,C 180,E1 -26887.823,E2 -26887.823} C_VEL
LIN {X 0,Y 94.06,Z 311.393,A -85,B 0,C 180,E1 -26897.041,E2 -26897.041} C_VEL
LIN {X 0,Y 94.189,Z 311.381,A -85,B 0,C 180,E1 -26901.412,E2 -26901.412} C_VEL
LIN {X 0,Y 94.789,Z 311.299,A -85,B 0,C 180,E1 -26909.994,E2 -26909.994} C_VEL
LIN {X 0,Y 94.193,Z 311.373,A -85,B 0,C 180,E1 -26918.576,E2 -26918.576} C_VEL
LIN {X 0,Y 94.034,Z 311.397,A -85,B 0,C 180,E1 -26923.704,E2 -26923.704} C_VEL
LIN {X 0,Y 93.684,Z 311.44,A -85,B 0,C 180,E1 -26932.023,E2 -26932.023} C_VEL
LIN {X 0,Y 93.611,Z 311.442,A -85,B 0,C 180,E1 -26936.766,E2 -26936.766} C_VEL
LIN {X 0,Y 93.586,Z 311.447,A -85,B 0,C 180,E1 -26944.31,E2 -26944.31} C_VEL
LIN {X 0,Y 93.526,Z 311.455,A -85,B 0,C 180,E1 -26952.547,E2 -26952.547} C_VEL
LIN {X 0,Y 93.521,Z 311.461,A -85,B 0,C 180,E1 -26958.71,E2 -26958.71} C_VEL
LIN {X 0,Y 93.575,Z 311.454,A -85,B 0,C 180,E1 -26965.695,E2 -26965.695} C_VEL
LIN {X 0,Y 93.657,Z 311.443,A -85,B 0,C 180,E1 -26974.206,E2 -26974.206} C_VEL
LIN {X 0,Y 93.681,Z 311.436,A -85,B 0,C 180,E1 -26977.973,E2 -26977.973} C_VEL
LIN {X 0,Y 94.08,Z 311.384,A -85,B 0,C 180,E1 -26987.053,E2 -26987.053} C_VEL
LIN {X 0,Y 94.189,Z 311.378,A -85,B 0,C 180,E1 -26991.421,E2 -26991.421} C_VEL
LIN {X 0,Y 94.785,Z 311.302,A -85,B 0,C 180,E1 -27000.003,E2 -27000.003} C_VEL
LIN {X 0,Y 94.191,Z 311.377,A -85,B 0,C 180,E1 -27008.586,E2 -27008.586} C_VEL
LIN {X 0,Y 94.034,Z 311.398,A -85,B 0,C 180,E1 -27013.714,E2 -27013.714} C_VEL
LIN {X 0,Y 93.799,Z 311.6,A -85,B 0,C 180,E1 -27020.279,E2 -27020.279} C_VEL
LIN {X 0,Y 94.937,Z 314.552,A -85,B 0,C 180,E1 -27021.3,E2 -27021.3} C_VEL
LIN {X 0,Y 97.083,Z 318.482,A -85,B 0,C 180,E1 -27022.849,E2 -27022.849} C_VEL
LIN {X 0,Y 103.435,Z 332.002,A -85,B 0,C 180,E1 -27027.302,E2 -27027.302} C_VEL
LIN {X 0,Y 107.557,Z 342.213,A -85,B 0,C 180,E1 -27030.098,E2 -27030.098} C_VEL
LIN {X 0,Y 115.767,Z 368.051,A -85,B 0,C 180,E1 -27035.758,E2 -27035.758} C_VEL
LIN {X 0,Y 121.515,Z 386.463,A -85,B 0,C 180,E1 -27039.244,E2 -27039.244} C_VEL
LIN {X 0,Y 110.738,Z 467.197,A -85,B 0,C 180,E1 -27048.371,E2 -27048.371} C_VEL
LIN {X 0,Y 108.229,Z 483.001,A -85,B 0,C 180,E1 -27050.949,E2 -27050.949} C_VEL
LIN {X 0,Y 105.361,Z 498.546,A -85,B 0,C 180,E1 -27054.298,E2 -27054.298} C_VEL
LIN {X 0,Y 102.425,Z 513.539,A -85,B 0,C 180,E1 -27058.46,E2 -27058.46} C_VEL
LIN {X 0,Y 100.04,Z 526.101,A -85,B 0,C 180,E1 -27062.836,E2 -27062.836} C_VEL
LIN {X 0,Y 97.659,Z 540.074,A -85,B 0,C 180,E1 -27068.917,E2 -27068.917} C_VEL
LIN {X 0,Y 96.28,Z 551.759,A -85,B 0,C 180,E1 -27075.204,E2 -27075.204} C_VEL
LIN {X 0,Y 95.908,Z 561.599,A -85,B 0,C 180,E1 -27081.578,E2 -27081.578} C_VEL
LIN {X 0,Y 96.276,Z 569.836,A -85,B 0,C 180,E1 -27087.914,E2 -27087.914} C_VEL
LIN {X 0,Y 96.699,Z 574.426,A -85,B 0,C 180,E1 -27092.088,E2 -27092.088} C_VEL
LIN {X 0,Y 96.814,Z 576.408,A -85,B 0,C 180,E1 -27094.169,E2 -27094.169} C_VEL
LIN {X 0,Y 96.426,Z 579.617,A -85,B 0,C 180,E1 -27098.388,E2 -27098.388} C_VEL
LIN {X 0,Y 96.385,Z 584.852,A -85,B 0,C 180,E1 -27106.963,E2 -27106.963} C_VEL
LIN {X 0,Y 100.376,Z 590.833,A -85,B 0,C 180,E1 -27119.354,E2 -27119.354} C_VEL
LIN {X 0,Y 109.205,Z 595.17,A -85,B 0,C 180,E1 -27130.064,E2 -27130.064} C_VEL
LIN {X 0,Y 117.149,Z 597.22,A -85,B 0,C 180,E1 -27136.052,E2 -27136.052} C_VEL
LIN {X 0,Y 118.11,Z 597.179,A -85,B 0,C 180,E1 -27137.82,E2 -27137.82} C_VEL
LIN {X 0,Y 108.849,Z 592.5,A -85,B 0,C 180,E1 -27144.469,E2 -27144.469} C_VEL
LIN {X 0,Y 101.117,Z 586.23,A -85,B 0,C 180,E1 -27153.139,E2 -27153.139} C_VEL
LIN {X 0,Y 96.101,Z 578.484,A -85,B 0,C 180,E1 -27162.988,E2 -27162.988} C_VEL
LIN {X 0,Y 94.071,Z 569.96,A -85,B 0,C 180,E1 -27172.484,E2 -27172.484} C_VEL
LIN {X 0,Y 93.548,Z 563.045,A -85,B 0,C 180,E1 -27178.92,E2 -27178.92} C_VEL
LIN {X 0,Y 93.466,Z 557.521,A -85,B 0,C 180,E1 -27183.435,E2 -27183.435} C_VEL
LIN {X 0,Y 92.97,Z 553.685,A -85,B 0,C 180,E1 -27186.142,E2 -27186.142} C_VEL
LIN {X 0,Y 91.687,Z 549.517,A -85,B 0,C 180,E1 -27188.672,E2 -27188.672} C_VEL
LIN {X 0,Y 88.848,Z 540.709,A -85,B 0,C 180,E1 -27193.496,E2 -27193.496} C_VEL
LIN {X 0,Y 88.306,Z 536.167,A -85,B 0,C 180,E1 -27196,E2 -27196} C_VEL
LIN {X 0,Y 88.396,Z 534.63,A -85,B 0,C 180,E1 -27196.848,E2 -27196.848} C_VEL
LIN {X 0,Y 90.487,Z 521.709,A -85,B 0,C 180,E1 -27203.452,E2 -27203.452} C_VEL
LIN {X 0,Y 93.282,Z 507.369,A -85,B 0,C 180,E1 -27209.318,E2 -27209.318} C_VEL
LIN {X 0,Y 96.462,Z 491.678,A -85,B 0,C 180,E1 -27214.373,E2 -27214.373} C_VEL
LIN {X 0,Y 99.801,Z 474.279,A -85,B 0,C 180,E1 -27218.597,E2 -27218.597} C_VEL
LIN {X 0,Y 102.643,Z 457.237,A -85,B 0,C 180,E1 -27221.711,E2 -27221.711} C_VEL
LIN {X 0,Y 106.614,Z 427.541,A -85,B 0,C 180,E1 -27225.624,E2 -27225.624} C_VEL
LIN {X 0,Y 113.814,Z 376.742,A -85,B 0,C 180,E1 -27231.421,E2 -27231.421} C_VEL
LIN {X 0,Y 104.258,Z 352.042,A -85,B 0,C 180,E1 -27237.221,E2 -27237.221} C_VEL
LIN {X 0,Y 97.489,Z 335.297,A -85,B 0,C 180,E1 -27241.989,E2 -27241.989} C_VEL
LIN {X 0,Y 91.507,Z 322.299,A -85,B 0,C 180,E1 -27246.598,E2 -27246.598} C_VEL
LIN {X 0,Y 88.038,Z 315.753,A -85,B 0,C 180,E1 -27249.399,E2 -27249.399} C_VEL
LIN {X 0,Y 86.806,Z 313.285,A -85,B 0,C 180,E1 -27250.484,E2 -27250.484} C_VEL
LIN {X 0,Y 86.635,Z 312.32,A -85,B 0,C 180,E1 -27250.905,E2 -27250.905} C_VEL
LIN {X 0,Y 86.928,Z 312.285,A -85,B 0,C 180,E1 -27255.957,E2 -27255.957} C_VEL
LIN {X 0,Y 87.094,Z 312.266,A -85,B 0,C 180,E1 -27260.706,E2 -27260.706} C_VEL
LIN {X 0,Y 87.716,Z 312.18,A -85,B 0,C 180,E1 -27269.994,E2 -27269.994} C_VEL
LIN {X 0,Y 87.101,Z 312.253,A -85,B 0,C 180,E1 -27279.28,E2 -27279.28} C_VEL
LIN {X 0,Y 86.942,Z 312.28,A -85,B 0,C 180,E1 -27284.082,E2 -27284.082} C_VEL
LIN {X 0,Y 86.578,Z 312.324,A -85,B 0,C 180,E1 -27293.939,E2 -27293.939} C_VEL
LIN {X 0,Y 86.466,Z 312.336,A -85,B 0,C 180,E1 -27299.181,E2 -27299.181} C_VEL
LIN {X 0,Y 86.505,Z 312.327,A -85,B 0,C 180,E1 -27305.672,E2 -27305.672} C_VEL
LIN {X 0,Y 86.468,Z 312.332,A -85,B 0,C 180,E1 -27312.993,E2 -27312.993} C_VEL
LIN {X 0,Y 86.443,Z 312.341,A -85,B 0,C 180,E1 -27319.432,E2 -27319.432} C_VEL
LIN {X 0,Y 86.518,Z 312.332,A -85,B 0,C 180,E1 -27325.35,E2 -27325.35} C_VEL
LIN {X 0,Y 86.572,Z 312.324,A -85,B 0,C 180,E1 -27333.236,E2 -27333.236} C_VEL
LIN {X 0,Y 86.635,Z 312.314,A -85,B 0,C 180,E1 -27341.069,E2 -27341.069} C_VEL
LIN {X 0,Y 86.959,Z 312.275,A -85,B 0,C 180,E1 -27345.972,E2 -27345.972} C_VEL
LIN {X 0,Y 87.097,Z 312.26,A -85,B 0,C 180,E1 -27350.717,E2 -27350.717} C_VEL
LIN {X 0,Y 87.712,Z 312.183,A -85,B 0,C 180,E1 -27360.004,E2 -27360.004} C_VEL
LIN {X 0,Y 87.099,Z 312.26,A -85,B 0,C 180,E1 -27369.291,E2 -27369.291} C_VEL
LIN {X 0,Y 86.942,Z 312.281,A -85,B 0,C 180,E1 -27374.092,E2 -27374.092} C_VEL
LIN {X 0,Y 86.767,Z 312.305,A -85,B 0,C 180,E1 -27377.063,E2 -27377.063} C_VEL
LIN {X 0,Y 87.788,Z 315.261,A -85,B 0,C 180,E1 -27378.265,E2 -27378.265} C_VEL
LIN {X 0,Y 90.816,Z 320.823,A -85,B 0,C 180,E1 -27380.716,E2 -27380.716} C_VEL
LIN {X 0,Y 96.725,Z 333.317,A -85,B 0,C 180,E1 -27385.273,E2 -27385.273} C_VEL
LIN {X 0,Y 101.184,Z 344.159,A -85,B 0,C 180,E1 -27388.559,E2 -27388.559} C_VEL
LIN {X 0,Y 108.733,Z 368.232,A -85,B 0,C 180,E1 -27394.234,E2 -27394.234} C_VEL
LIN {X 0,Y 114.657,Z 387.606,A -85,B 0,C 180,E1 -27398.163,E2 -27398.163} C_VEL
LIN {X 0,Y 103.799,Z 466.467,A -85,B 0,C 180,E1 -27407.674,E2 -27407.674} C_VEL
LIN {X 0,Y 101.211,Z 482.411,A -85,B 0,C 180,E1 -27410.436,E2 -27410.436} C_VEL
LIN {X 0,Y 98.388,Z 497.462,A -85,B 0,C 180,E1 -27413.899,E2 -27413.899} C_VEL
LIN {X 0,Y 95.437,Z 512.453,A -85,B 0,C 180,E1 -27418.36,E2 -27418.36} C_VEL
LIN {X 0,Y 92.796,Z 526.286,A -85,B 0,C 180,E1 -27423.587,E2 -27423.587} C_VEL
LIN {X 0,Y 90.718,Z 538.936,A -85,B 0,C 180,E1 -27429.584,E2 -27429.584} C_VEL
LIN {X 0,Y 89.489,Z 550.666,A -85,B 0,C 180,E1 -27436.379,E2 -27436.379} C_VEL
LIN {X 0,Y 89.29,Z 560.458,A -85,B 0,C 180,E1 -27443.226,E2 -27443.226} C_VEL
LIN {X 0,Y 89.936,Z 568.692,A -85,B 0,C 180,E1 -27450.006,E2 -27450.006} C_VEL
LIN {X 0,Y 90.36,Z 573.135,A -85,B 0,C 180,E1 -27454.467,E2 -27454.467} C_VEL
LIN {X 0,Y 90.344,Z 574.951,A -85,B 0,C 180,E1 -27456.707,E2 -27456.707} C_VEL
LIN {X 0,Y 89.984,Z 580.733,A -85,B 0,C 180,E1 -27465.87,E2 -27465.87} C_VEL
LIN {X 0,Y 92.543,Z 586.344,A -85,B 0,C 180,E1 -27477.114,E2 -27477.114} C_VEL
LIN {X 0,Y 97.307,Z 590.013,A -85,B 0,C 180,E1 -27485.302,E2 -27485.302} C_VEL
LIN {X 0,Y 104.108,Z 592.955,A -85,B 0,C 180,E1 -27492.466,E2 -27492.466} C_VEL
LIN {X 0,Y 109.21,Z 594.486,A -85,B 0,C 180,E1 -27496.427,E2 -27496.427} C_VEL
LIN {X 0,Y 108.952,Z 594.114,A -85,B 0,C 180,E1 -27497.97,E2 -27497.97} C_VEL
LIN {X 0,Y 99.654,Z 588.449,A -85,B 0,C 180,E1 -27505.65,E2 -27505.65} C_VEL
LIN {X 0,Y 92.545,Z 581.234,A -85,B 0,C 180,E1 -27515.311,E2 -27515.311} C_VEL
LIN {X 0,Y 88.979,Z 574.346,A -85,B 0,C 180,E1 -27523.948,E2 -27523.948} C_VEL
LIN {X 0,Y 87.476,Z 567.266,A -85,B 0,C 180,E1 -27531.914,E2 -27531.914} C_VEL
LIN {X 0,Y 86.867,Z 560.074,A -85,B 0,C 180,E1 -27538.837,E2 -27538.837} C_VEL
LIN {X 0,Y 86.868,Z 551.538,A -85,B 0,C 180,E1 -27545.801,E2 -27545.801} C_VEL
LIN {X 0,Y 87.773,Z 539.659,A -85,B 0,C 180,E1 -27553.895,E2 -27553.895} C_VEL
LIN {X 0,Y 88.396,Z 534.63,A -85,B 0,C 180,E1 -27556.848,E2 -27556.848} C_VEL
LIN {X 0,Y 88.343,Z 530.065,A -85,B 0,C 180,E1 -27559.246,E2 -27559.246} C_VEL
LIN {X 0,Y 86.81,Z 522.055,A -85,B 0,C 180,E1 -27562.915,E2 -27562.915} C_VEL
LIN {X 0,Y 85.489,Z 513.752,A -85,B 0,C 180,E1 -27566.479,E2 -27566.479} C_VEL
LIN {X 0,Y 85.819,Z 508.648,A -85,B 0,C 180,E1 -27568.57,E2 -27568.57} C_VEL
LIN {X 0,Y 88.698,Z 494.438,A -85,B 0,C 180,E1 -27573.682,E2 -27573.682} C_VEL
LIN {X 0,Y 92.047,Z 477.892,A -85,B 0,C 180,E1 -27578.292,E2 -27578.292} C_VEL
LIN {X 0,Y 95.204,Z 460.023,A -85,B 0,C 180,E1 -27581.981,E2 -27581.981} C_VEL
LIN {X 0,Y 98.338,Z 438.19,A -85,B 0,C 180,E1 -27585.21,E2 -27585.21} C_VEL
LIN {X 0,Y 106.956,Z 378.063,A -85,B 0,C 180,E1 -27592.68,E2 -27592.68} C_VEL
LIN {X 0,Y 97.168,Z 352.244,A -85,B 0,C 180,E1 -27599.238,E2 -27599.238} C_VEL
LIN {X 0,Y 90.664,Z 336.176,A -85,B 0,C 180,E1 -27604.317,E2 -27604.317} C_VEL
LIN {X 0,Y 84.94,Z 323.817,A -85,B 0,C 180,E1 -27609.247,E2 -27609.247} C_VEL
LIN {X 0,Y 81.011,Z 316.563,A -85,B 0,C 180,E1 -27612.829,E2 -27612.829} C_VEL
LIN {X 0,Y 79.846,Z 313.96,A -85,B 0,C 180,E1 -27614.101,E2 -27614.101} C_VEL
LIN {X 0,Y 79.72,Z 313.186,A -85,B 0,C 180,E1 -27614.433,E2 -27614.433} C_VEL
LIN {X 0,Y 79.973,Z 313.153,A -85,B 0,C 180,E1 -27619.87,E2 -27619.87} C_VEL
LIN {X 0,Y 80.644,Z 313.061,A -85,B 0,C 180,E1 -27629.993,E2 -27629.993} C_VEL
LIN {X 0,Y 79.986,Z 313.138,A -85,B 0,C 180,E1 -27640.114,E2 -27640.114} C_VEL
LIN {X 0,Y 79.754,Z 313.175,A -85,B 0,C 180,E1 -27645.322,E2 -27645.322} C_VEL
LIN {X 0,Y 79.505,Z 313.204,A -85,B 0,C 180,E1 -27650.699,E2 -27650.699} C_VEL
LIN {X 0,Y 79.472,Z 313.203,A -85,B 0,C 180,E1 -27657.84,E2 -27657.84} C_VEL
LIN {X 0,Y 79.372,Z 313.222,A -85,B 0,C 180,E1 -27662.083,E2 -27662.083} C_VEL
LIN {X 0,Y 79.361,Z 313.223,A -85,B 0,C 180,E1 -27668.3,E2 -27668.3} C_VEL
LIN {X 0,Y 79.374,Z 313.216,A -85,B 0,C 180,E1 -27675.089,E2 -27675.089} C_VEL
LIN {X 0,Y 79.373,Z 313.215,A -85,B 0,C 180,E1 -27682.823,E2 -27682.823} C_VEL
LIN {X 0,Y 79.365,Z 313.223,A -85,B 0,C 180,E1 -27687.91,E2 -27687.91} C_VEL
LIN {X 0,Y 79.513,Z 313.205,A -85,B 0,C 180,E1 -27693.777,E2 -27693.777} C_VEL
LIN {X 0,Y 79.502,Z 313.199,A -85,B 0,C 180,E1 -27699.297,E2 -27699.297} C_VEL
LIN {X 0,Y 79.83,Z 313.163,A -85,B 0,C 180,E1 -27705.528,E2 -27705.528} C_VEL
LIN {X 0,Y 79.982,Z 313.145,A -85,B 0,C 180,E1 -27709.882,E2 -27709.882} C_VEL
LIN {X 0,Y 80.64,Z 313.064,A -85,B 0,C 180,E1 -27720.004,E2 -27720.004} C_VEL
LIN {X 0,Y 79.984,Z 313.145,A -85,B 0,C 180,E1 -27730.125,E2 -27730.125} C_VEL
LIN {X 0,Y 79.959,Z 313.347,A -85,B 0,C 180,E1 -27733.7,E2 -27733.7} C_VEL
LIN {X 0,Y 80.939,Z 316.209,A -85,B 0,C 180,E1 -27734.921,E2 -27734.921} C_VEL
LIN {X 0,Y 85.433,Z 324.674,A -85,B 0,C 180,E1 -27739.059,E2 -27739.059} C_VEL
LIN {X 0,Y 91.546,Z 337.968,A -85,B 0,C 180,E1 -27744.223,E2 -27744.223} C_VEL
LIN {X 0,Y 95.409,Z 347.77,A -85,B 0,C 180,E1 -27747.339,E2 -27747.339} C_VEL
LIN {X 0,Y 103.013,Z 372.611,A -85,B 0,C 180,E1 -27753.521,E2 -27753.521} C_VEL
LIN {X 0,Y 107.859,Z 388.804,A -85,B 0,C 180,E1 -27757.018,E2 -27757.018} C_VEL
LIN {X 0,Y 96.877,Z 465.728,A -85,B 0,C 180,E1 -27766.927,E2 -27766.927} C_VEL
LIN {X 0,Y 94.172,Z 481.914,A -85,B 0,C 180,E1 -27769.942,E2 -27769.942} C_VEL
LIN {X 0,Y 91.101,Z 498.02,A -85,B 0,C 180,E1 -27773.976,E2 -27773.976} C_VEL
LIN {X 0,Y 88.456,Z 511.215,A -85,B 0,C 180,E1 -27778.247,E2 -27778.247} C_VEL
LIN {X 0,Y 85.974,Z 524.309,A -85,B 0,C 180,E1 -27783.551,E2 -27783.551} C_VEL
LIN {X 0,Y 83.814,Z 537.77,A -85,B 0,C 180,E1 -27790.41,E2 -27790.41} C_VEL
LIN {X 0,Y 82.773,Z 549.449,A -85,B 0,C 180,E1 -27797.752,E2 -27797.752} C_VEL
LIN {X 0,Y 82.82,Z 559.252,A -85,B 0,C 180,E1 -27805.139,E2 -27805.139} C_VEL
LIN {X 0,Y 83.744,Z 567.401,A -85,B 0,C 180,E1 -27812.411,E2 -27812.411} C_VEL
LIN {X 0,Y 84.029,Z 569.652,A -85,B 0,C 180,E1 -27814.804,E2 -27814.804} C_VEL
LIN {X 0,Y 84.059,Z 571.605,A -85,B 0,C 180,E1 -27817.211,E2 -27817.211} C_VEL
LIN {X 0,Y 83.743,Z 576.276,A -85,B 0,C 180,E1 -27824.589,E2 -27824.589} C_VEL
LIN {X 0,Y 85.333,Z 581.639,A -85,B 0,C 180,E1 -27835.04,E2 -27835.04} C_VEL
LIN {X 0,Y 91.996,Z 587.39,A -85,B 0,C 180,E1 -27847.68,E2 -27847.68} C_VEL
LIN {X 0,Y 100.51,Z 590.982,A -85,B 0,C 180,E1 -27856.073,E2 -27856.073} C_VEL
LIN {X 0,Y 100.909,Z 590.945,A -85,B 0,C 180,E1 -27857.475,E2 -27857.475} C_VEL
LIN {X 0,Y 90.752,Z 583.723,A -85,B 0,C 180,E1 -27867.17,E2 -27867.17} C_VEL
LIN {X 0,Y 84.042,Z 575.007,A -85,B 0,C 180,E1 -27878.639,E2 -27878.639} C_VEL
LIN {X 0,Y 81.117,Z 565.532,A -85,B 0,C 180,E1 -27890.018,E2 -27890.018} C_VEL
LIN {X 0,Y 80.324,Z 558.174,A -85,B 0,C 180,E1 -27897.489,E2 -27897.489} C_VEL
LIN {X 0,Y 80.164,Z 549.471,A -85,B 0,C 180,E1 -27905.026,E2 -27905.026} C_VEL
LIN {X 0,Y 81.013,Z 537.256,A -85,B 0,C 180,E1 -27913.798,E2 -27913.798} C_VEL
LIN {X 0,Y 82.663,Z 525.112,A -85,B 0,C 180,E1 -27920.93,E2 -27920.93} C_VEL
LIN {X 0,Y 85.327,Z 511.008,A -85,B 0,C 180,E1 -27927.596,E2 -27927.596} C_VEL
LIN {X 0,Y 85.819,Z 508.648,A -85,B 0,C 180,E1 -27928.57,E2 -27928.57} C_VEL
LIN {X 0,Y 86.146,Z 503.562,A -85,B 0,C 180,E1 -27930.536,E2 -27930.536} C_VEL
LIN {X 0,Y 84.964,Z 494.847,A -85,B 0,C 180,E1 -27933.588,E2 -27933.588} C_VEL
LIN {X 0,Y 83.882,Z 485.924,A -85,B 0,C 180,E1 -27936.493,E2 -27936.493} C_VEL
LIN {X 0,Y 84.382,Z 480.417,A -85,B 0,C 180,E1 -27938.079,E2 -27938.079} C_VEL
LIN {X 0,Y 87.472,Z 464.338,A -85,B 0,C 180,E1 -27941.898,E2 -27941.898} C_VEL
LIN {X 0,Y 90.304,Z 446.025,A -85,B 0,C 180,E1 -27945.064,E2 -27945.064} C_VEL
LIN {X 0,Y 100.18,Z 379.535,A -85,B 0,C 180,E1 -27953.989,E2 -27953.989} C_VEL
LIN {X 0,Y 91.232,Z 355.468,A -85,B 0,C 180,E1 -27960.581,E2 -27960.581} C_VEL
LIN {X 0,Y 85.162,Z 340.033,A -85,B 0,C 180,E1 -27965.794,E2 -27965.794} C_VEL
LIN {X 0,Y 79.68,Z 327.949,A -85,B 0,C 180,E1 -27970.977,E2 -27970.977} C_VEL
LIN {X 0,Y 75.548,Z 320.077,A -85,B 0,C 180,E1 -27975.244,E2 -27975.244} C_VEL
LIN {X 0,Y 74.444,Z 317.793,A -85,B 0,C 180,E1 -27976.535,E2 -27976.535} C_VEL
LIN {X 0,Y 73.077,Z 315.221,A -85,B 0,C 180,E1 -27978.156,E2 -27978.156} C_VEL
LIN {X 0,Y 72.861,Z 314.037,A -85,B 0,C 180,E1 -27978.869,E2 -27978.869} C_VEL
LIN {X 0,Y 73.57,Z 313.942,A -85,B 0,C 180,E1 -27989.993,E2 -27989.993} C_VEL
LIN {X 0,Y 72.872,Z 314.025,A -85,B 0,C 180,E1 -28001.113,E2 -28001.113} C_VEL
LIN {X 0,Y 72.574,Z 314.065,A -85,B 0,C 180,E1 -28006.881,E2 -28006.881} C_VEL
LIN {X 0,Y 72.385,Z 314.094,A -85,B 0,C 180,E1 -28012.845,E2 -28012.845} C_VEL
LIN {X 0,Y 72.367,Z 314.092,A -85,B 0,C 180,E1 -28019.078,E2 -28019.078} C_VEL
LIN {X 0,Y 72.288,Z 314.097,A -85,B 0,C 180,E1 -28025.675,E2 -28025.675} C_VEL
LIN {X 0,Y 72.236,Z 314.105,A -85,B 0,C 180,E1 -28032.914,E2 -28032.914} C_VEL
LIN {X 0,Y 72.281,Z 314.1,A -85,B 0,C 180,E1 -28041.052,E2 -28041.052} C_VEL
LIN {X 0,Y 72.281,Z 314.103,A -85,B 0,C 180,E1 -28044.316,E2 -28044.316} C_VEL
LIN {X 0,Y 72.363,Z 314.088,A -85,B 0,C 180,E1 -28050.953,E2 -28050.953} C_VEL
LIN {X 0,Y 72.382,Z 314.09,A -85,B 0,C 180,E1 -28057.151,E2 -28057.151} C_VEL
LIN {X 0,Y 72.725,Z 314.049,A -85,B 0,C 180,E1 -28065.069,E2 -28065.069} C_VEL
LIN {X 0,Y 72.869,Z 314.026,A -85,B 0,C 180,E1 -28068.883,E2 -28068.883} C_VEL
LIN {X 0,Y 73.567,Z 313.945,A -85,B 0,C 180,E1 -28080.004,E2 -28080.004} C_VEL
LIN {X 0,Y 72.93,Z 314.025,A -85,B 0,C 180,E1 -28089.188,E2 -28089.188} C_VEL
LIN {X 0,Y 74.117,Z 317.176,A -85,B 0,C 180,E1 -28090.936,E2 -28090.936} C_VEL
LIN {X 0,Y 75.262,Z 318.963,A -85,B 0,C 180,E1 -28092.145,E2 -28092.145} C_VEL
LIN {X 0,Y 81.25,Z 330.974,A -85,B 0,C 180,E1 -28098.343,E2 -28098.343} C_VEL
LIN {X 0,Y 86.597,Z 343.28,A -85,B 0,C 180,E1 -28103.315,E2 -28103.315} C_VEL
LIN {X 0,Y 89.634,Z 351.394,A -85,B 0,C 180,E1 -28106.018,E2 -28106.018} C_VEL
LIN {X 0,Y 96.899,Z 375.787,A -85,B 0,C 180,E1 -28112.495,E2 -28112.495} C_VEL
LIN {X 0,Y 101.021,Z 389.845,A -85,B 0,C 180,E1 -28115.737,E2 -28115.737} C_VEL
LIN {X 0,Y 89.947,Z 464.911,A -85,B 0,C 180,E1 -28126.106,E2 -28126.106} C_VEL
LIN {X 0,Y 87.134,Z 481.488,A -85,B 0,C 180,E1 -28129.444,E2 -28129.444} C_VEL
LIN {X 0,Y 83.852,Z 498.339,A -85,B 0,C 180,E1 -28134.086,E2 -28134.086} C_VEL
LIN {X 0,Y 80.896,Z 512.764,A -85,B 0,C 180,E1 -28139.319,E2 -28139.319} C_VEL
LIN {X 0,Y 78.551,Z 525.64,A -85,B 0,C 180,E1 -28145.264,E2 -28145.264} C_VEL
LIN {X 0,Y 76.758,Z 538.557,A -85,B 0,C 180,E1 -28152.696,E2 -28152.696} C_VEL
LIN {X 0,Y 76.115,Z 549.875,A -85,B 0,C 180,E1 -28160.709,E2 -28160.709} C_VEL
LIN {X 0,Y 76.663,Z 559.391,A -85,B 0,C 180,E1 -28168.694,E2 -28168.694} C_VEL
LIN {X 0,Y 77.691,Z 565.963,A -85,B 0,C 180,E1 -28175.197,E2 -28175.197} C_VEL
LIN {X 0,Y 77.838,Z 568.096,A -85,B 0,C 180,E1 -28177.788,E2 -28177.788} C_VEL
LIN {X 0,Y 77.683,Z 572.952,A -85,B 0,C 180,E1 -28185.755,E2 -28185.755} C_VEL
LIN {X 0,Y 80.13,Z 579.346,A -85,B 0,C 180,E1 -28198.702,E2 -28198.702} C_VEL
LIN {X 0,Y 86.903,Z 584.584,A -85,B 0,C 180,E1 -28210.321,E2 -28210.321} C_VEL
LIN {X 0,Y 90.568,Z 586.381,A -85,B 0,C 180,E1 -28214.306,E2 -28214.306} C_VEL
LIN {X 0,Y 92.875,Z 587.221,A -85,B 0,C 180,E1 -28217.07,E2 -28217.07} C_VEL
LIN {X 0,Y 83.353,Z 579.693,A -85,B 0,C 180,E1 -28227.05,E2 -28227.05} C_VEL
LIN {X 0,Y 77.231,Z 570.983,A -85,B 0,C 180,E1 -28238.65,E2 -28238.65} C_VEL
LIN {X 0,Y 74.699,Z 562.471,A -85,B 0,C 180,E1 -28249.15,E2 -28249.15} C_VEL
LIN {X 0,Y 73.766,Z 554.746,A -85,B 0,C 180,E1 -28257.265,E2 -28257.265} C_VEL
LIN {X 0,Y 73.511,Z 547.197,A -85,B 0,C 180,E1 -28264.108,E2 -28264.108} C_VEL
LIN {X 0,Y 74.292,Z 534.672,A -85,B 0,C 180,E1 -28273.676,E2 -28273.676} C_VEL
LIN {X 0,Y 75.759,Z 523.628,A -85,B 0,C 180,E1 -28280.581,E2 -28280.581} C_VEL
LIN {X 0,Y 78.526,Z 508.983,A -85,B 0,C 180,E1 -28288.021,E2 -28288.021} C_VEL
LIN {X 0,Y 81.653,Z 493.696,A -85,B 0,C 180,E1 -28294.014,E2 -28294.014} C_VEL
LIN {X 0,Y 84.382,Z 480.417,A -85,B 0,C 180,E1 -28298.079,E2 -28298.079} C_VEL
LIN {X 0,Y 84.862,Z 474.973,A -85,B 0,C 180,E1 -28299.553,E2 -28299.553} C_VEL
LIN {X 0,Y 83.736,Z 465.795,A -85,B 0,C 180,E1 -28301.932,E2 -28301.932} C_VEL
LIN {X 0,Y 82.654,Z 458.294,A -85,B 0,C 180,E1 -28303.747,E2 -28303.747} C_VEL
LIN {X 0,Y 82.457,Z 452.595,A -85,B 0,C 180,E1 -28304.944,E2 -28304.944} C_VEL
LIN {X 0,Y 82.651,Z 450.661,A -85,B 0,C 180,E1 -28305.297,E2 -28305.297} C_VEL
LIN {X 0,Y 93.374,Z 380.812,A -85,B 0,C 180,E1 -28315.478,E2 -28315.478} C_VEL
LIN {X 0,Y 85.18,Z 358.363,A -85,B 0,C 180,E1 -28322.147,E2 -28322.147} C_VEL
LIN {X 0,Y 79.641,Z 343.773,A -85,B 0,C 180,E1 -28327.453,E2 -28327.453} C_VEL
LIN {X 0,Y 74.535,Z 332.152,A -85,B 0,C 180,E1 -28332.854,E2 -28332.854} C_VEL
LIN {X 0,Y 69.509,Z 322.153,A -85,B 0,C 180,E1 -28338.879,E2 -28338.879} C_VEL
LIN {X 0,Y 67.868,Z 319.061,A -85,B 0,C 180,E1 -28341.056,E2 -28341.056} C_VEL
LIN {X 0,Y 66.322,Z 316.598,A -85,B 0,C 180,E1 -28343.145,E2 -28343.145} C_VEL
LIN {X 0,Y 65.972,Z 314.888,A -85,B 0,C 180,E1 -28344.26,E2 -28344.26} C_VEL
LIN {X 0,Y 66.494,Z 314.822,A -85,B 0,C 180,E1 -28349.992,E2 -28349.992} C_VEL
LIN {X 0,Y 65.765,Z 314.914,A -85,B 0,C 180,E1 -28362.332,E2 -28362.332} C_VEL
LIN {X 0,Y 65.376,Z 314.957,A -85,B 0,C 180,E1 -28368.805,E2 -28368.805} C_VEL
LIN {X 0,Y 65.228,Z 314.979,A -85,B 0,C 180,E1 -28375.52,E2 -28375.52} C_VEL
LIN {X 0,Y 65.187,Z 314.989,A -85,B 0,C 180,E1 -28382.609,E2 -28382.609} C_VEL
LIN {X 0,Y 65.174,Z 314.99,A -85,B 0,C 180,E1 -28390.996,E2 -28390.996} C_VEL
LIN {X 0,Y 65.189,Z 314.988,A -85,B 0,C 180,E1 -28399.701,E2 -28399.701} C_VEL
LIN {X 0,Y 65.242,Z 314.976,A -85,B 0,C 180,E1 -28409.499,E2 -28409.499} C_VEL
LIN {X 0,Y 65.228,Z 314.985,A -85,B 0,C 180,E1 -28414.476,E2 -28414.476} C_VEL
LIN {X 0,Y 65.625,Z 314.935,A -85,B 0,C 180,E1 -28424.511,E2 -28424.511} C_VEL
LIN {X 0,Y 65.762,Z 314.909,A -85,B 0,C 180,E1 -28427.663,E2 -28427.663} C_VEL
LIN {X 0,Y 66.491,Z 314.827,A -85,B 0,C 180,E1 -28440.005,E2 -28440.005} C_VEL
LIN {X 0,Y 66.104,Z 315.031,A -85,B 0,C 180,E1 -28444.006,E2 -28444.006} C_VEL
LIN {X 0,Y 66.995,Z 317.75,A -85,B 0,C 180,E1 -28445.649,E2 -28445.649} C_VEL
LIN {X 0,Y 68.643,Z 320.169,A -85,B 0,C 180,E1 -28447.727,E2 -28447.727} C_VEL
LIN {X 0,Y 71.922,Z 326.586,A -85,B 0,C 180,E1 -28451.916,E2 -28451.916} C_VEL
LIN {X 0,Y 76.315,Z 335.896,A -85,B 0,C 180,E1 -28456.902,E2 -28456.902} C_VEL
LIN {X 0,Y 81.015,Z 346.999,A -85,B 0,C 180,E1 -28461.713,E2 -28461.713} C_VEL
LIN {X 0,Y 83.7,Z 354.416,A -85,B 0,C 180,E1 -28464.385,E2 -28464.385} C_VEL
LIN {X 0,Y 90.583,Z 378.228,A -85,B 0,C 180,E1 -28471.199,E2 -28471.199} C_VEL
LIN {X 0,Y 94.212,Z 390.754,A -85,B 0,C 180,E1 -28474.317,E2 -28474.317} C_VEL
LIN {X 0,Y 82.995,Z 464.335,A -85,B 0,C 180,E1 -28485.269,E2 -28485.269} C_VEL
LIN {X 0,Y 80.113,Z 480.84,A -85,B 0,C 180,E1 -28488.867,E2 -28488.867} C_VEL
LIN {X 0,Y 76.978,Z 496.716,A -85,B 0,C 180,E1 -28493.608,E2 -28493.608} C_VEL
LIN {X 0,Y 73.898,Z 511.735,A -85,B 0,C 180,E1 -28499.534,E2 -28499.534} C_VEL
LIN {X 0,Y 71.543,Z 524.825,A -85,B 0,C 180,E1 -28506.2,E2 -28506.2} C_VEL
LIN {X 0,Y 69.886,Z 538.093,A -85,B 0,C 180,E1 -28514.702,E2 -28514.702} C_VEL
LIN {X 0,Y 69.705,Z 550.153,A -85,B 0,C 180,E1 -28524.221,E2 -28524.221} C_VEL
LIN {X 0,Y 70.766,Z 559.334,A -85,B 0,C 180,E1 -28532.854,E2 -28532.854} C_VEL
LIN {X 0,Y 71.599,Z 563.24,A -85,B 0,C 180,E1 -28537.024,E2 -28537.024} C_VEL
LIN {X 0,Y 71.729,Z 566.404,A -85,B 0,C 180,E1 -28541.518,E2 -28541.518} C_VEL
LIN {X 0,Y 72.389,Z 572.321,A -85,B 0,C 180,E1 -28552.86,E2 -28552.86} C_VEL
LIN {X 0,Y 77.167,Z 578.493,A -85,B 0,C 180,E1 -28566.307,E2 -28566.307} C_VEL
LIN {X 0,Y 83.635,Z 582.433,A -85,B 0,C 180,E1 -28574.971,E2 -28574.971} C_VEL
LIN {X 0,Y 84.856,Z 582.931,A -85,B 0,C 180,E1 -28576.708,E2 -28576.708} C_VEL
LIN {X 0,Y 76.394,Z 575.586,A -85,B 0,C 180,E1 -28586.492,E2 -28586.492} C_VEL
LIN {X 0,Y 70.704,Z 567.048,A -85,B 0,C 180,E1 -28598.11,E2 -28598.11} C_VEL
LIN {X 0,Y 68.363,Z 559.178,A -85,B 0,C 180,E1 -28608.13,E2 -28608.13} C_VEL
LIN {X 0,Y 67.376,Z 552.52,A -85,B 0,C 180,E1 -28615.508,E2 -28615.508} C_VEL
LIN {X 0,Y 66.932,Z 544.775,A -85,B 0,C 180,E1 -28623.005,E2 -28623.005} C_VEL
LIN {X 0,Y 67.619,Z 531.896,A -85,B 0,C 180,E1 -28633.519,E2 -28633.519} C_VEL
LIN {X 0,Y 69.558,Z 518.116,A -85,B 0,C 180,E1 -28642.512,E2 -28642.512} C_VEL
LIN {X 0,Y 72.36,Z 503.819,A -85,B 0,C 180,E1 -28649.847,E2 -28649.847} C_VEL
LIN {X 0,Y 75.767,Z 487.533,A -85,B 0,C 180,E1 -28656.246,E2 -28656.246} C_VEL
LIN {X 0,Y 79.043,Z 471.466,A -85,B 0,C 180,E1 -28660.97,E2 -28660.97} C_VEL
LIN {X 0,Y 81.997,Z 454.83,A -85,B 0,C 180,E1 -28664.562,E2 -28664.562} C_VEL
LIN {X 0,Y 82.651,Z 450.661,A -85,B 0,C 180,E1 -28665.297,E2 -28665.297} C_VEL
LIN {X 0,Y 82.824,Z 444.957,A -85,B 0,C 180,E1 -28666.376,E2 -28666.376} C_VEL
LIN {X 0,Y 79.988,Z 426.157,A -85,B 0,C 180,E1 -28670.443,E2 -28670.443} C_VEL
LIN {X 0,Y 80.284,Z 420.433,A -85,B 0,C 180,E1 -28671.486,E2 -28671.486} C_VEL
LIN {X 0,Y 86.592,Z 382.06,A -85,B 0,C 180,E1 -28677.151,E2 -28677.151} C_VEL
LIN {X 0,Y 78.335,Z 358.829,A -85,B 0,C 180,E1 -28684.768,E2 -28684.768} C_VEL
LIN {X 0,Y 73.363,Z 345.602,A -85,B 0,C 180,E1 -28690.213,E2 -28690.213} C_VEL
LIN {X 0,Y 68.451,Z 334.154,A -85,B 0,C 180,E1 -28696.257,E2 -28696.257} C_VEL
LIN {X 0,Y 64.297,Z 325.666,A -85,B 0,C 180,E1 -28702.081,E2 -28702.081} C_VEL
LIN {X 0,Y 61.665,Z 320.602,A -85,B 0,C 180,E1 -28706.315,E2 -28706.315} C_VEL
LIN {X 0,Y 59.896,Z 317.71,A -85,B 0,C 180,E1 -28709.361,E2 -28709.361} C_VEL
LIN {X 0,Y 59.27,Z 315.719,A -85,B 0,C 180,E1 -28711.052,E2 -28711.052} C_VEL
LIN {X 0,Y 58.638,Z 315.806,A -85,B 0,C 180,E1 -28723.859,E2 -28723.859} C_VEL
LIN {X 0,Y 58.181,Z 315.861,A -85,B 0,C 180,E1 -28731.237,E2 -28731.237} C_VEL
LIN {X 0,Y 58.14,Z 315.863,A -85,B 0,C 180,E1 -28738.904,E2 -28738.904} C_VEL
LIN {X 0,Y 58.149,Z 315.866,A -85,B 0,C 180,E1 -28742.228,E2 -28742.228} C_VEL
LIN {X 0,Y 58.022,Z 315.877,A -85,B 0,C 180,E1 -28747.262,E2 -28747.262} C_VEL
LIN {X 0,Y 58,Z 315.883,A -85,B 0,C 180,E1 -28756.624,E2 -28756.624} C_VEL
LIN {X 0,Y 58.018,Z 315.874,A -85,B 0,C 180,E1 -28762.73,E2 -28762.73} C_VEL
LIN {X 0,Y 58.145,Z 315.866,A -85,B 0,C 180,E1 -28767.77,E2 -28767.77} C_VEL
LIN {X 0,Y 58.138,Z 315.859,A -85,B 0,C 180,E1 -28771.09,E2 -28771.09} C_VEL
LIN {X 0,Y 58.515,Z 315.821,A -85,B 0,C 180,E1 -28783.879,E2 -28783.879} C_VEL
LIN {X 0,Y 58.806,Z 315.783,A -85,B 0,C 180,E1 -28793.142,E2 -28793.142} C_VEL
LIN {X 0,Y 59.02,Z 315.759,A -85,B 0,C 180,E1 -28796.592,E2 -28796.592} C_VEL
LIN {X 0,Y 60.234,Z 318.491,A -85,B 0,C 180,E1 -28799.17,E2 -28799.17} C_VEL
LIN {X 0,Y 61.8,Z 320.577,A -85,B 0,C 180,E1 -28801.636,E2 -28801.636} C_VEL
LIN {X 0,Y 63.575,Z 324.09,A -85,B 0,C 180,E1 -28804.604,E2 -28804.604} C_VEL
LIN {X 0,Y 66.95,Z 330.629,A -85,B 0,C 180,E1 -28809.445,E2 -28809.445} C_VEL
LIN {X 0,Y 71.594,Z 341.068,A -85,B 0,C 180,E1 -28815.482,E2 -28815.482} C_VEL
LIN {X 0,Y 76.606,Z 353.665,A -85,B 0,C 180,E1 -28821.18,E2 -28821.18} C_VEL
LIN {X 0,Y 80.96,Z 368.723,A -85,B 0,C 180,E1 -28826.247,E2 -28826.247} C_VEL
LIN {X 0,Y 87.446,Z 391.962,A -85,B 0,C 180,E1 -28832.816,E2 -28832.816} C_VEL
LIN {X 0,Y 76.09,Z 463.431,A -85,B 0,C 180,E1 -28844.301,E2 -28844.301} C_VEL
LIN {X 0,Y 73.139,Z 479.955,A -85,B 0,C 180,E1 -28848.203,E2 -28848.203} C_VEL
LIN {X 0,Y 70.124,Z 494.936,A -85,B 0,C 180,E1 -28853.045,E2 -28853.045} C_VEL
LIN {X 0,Y 67.089,Z 509.516,A -85,B 0,C 180,E1 -28859.3,E2 -28859.3} C_VEL
LIN {X 0,Y 64.726,Z 523.092,A -85,B 0,C 180,E1 -28866.83,E2 -28866.83} C_VEL
LIN {X 0,Y 63.244,Z 536.522,A -85,B 0,C 180,E1 -28876.35,E2 -28876.35} C_VEL
LIN {X 0,Y 63.391,Z 548.03,A -85,B 0,C 180,E1 -28886.274,E2 -28886.274} C_VEL
LIN {X 0,Y 64.954,Z 557.797,A -85,B 0,C 180,E1 -28896.22,E2 -28896.22} C_VEL
LIN {X 0,Y 65.771,Z 561.332,A -85,B 0,C 180,E1 -28900.493,E2 -28900.493} C_VEL
LIN {X 0,Y 65.971,Z 565.838,A -85,B 0,C 180,E1 -28908.647,E2 -28908.647} C_VEL
LIN {X 0,Y 69.638,Z 572.95,A -85,B 0,C 180,E1 -28924.277,E2 -28924.277} C_VEL
LIN {X 0,Y 75.615,Z 577.413,A -85,B 0,C 180,E1 -28934.203,E2 -28934.203} C_VEL
LIN {X 0,Y 76.8,Z 577.987,A -85,B 0,C 180,E1 -28936.658,E2 -28936.658} C_VEL
LIN {X 0,Y 67.925,Z 569.009,A -85,B 0,C 180,E1 -28948.841,E2 -28948.841} C_VEL
LIN {X 0,Y 63.114,Z 559.371,A -85,B 0,C 180,E1 -28962.163,E2 -28962.163} C_VEL
LIN {X 0,Y 61.357,Z 551.617,A -85,B 0,C 180,E1 -28971.763,E2 -28971.763} C_VEL
LIN {X 0,Y 60.566,Z 543.862,A -85,B 0,C 180,E1 -28979.995,E2 -28979.995} C_VEL
LIN {X 0,Y 60.74,Z 531.981,A -85,B 0,C 180,E1 -28990.832,E2 -28990.832} C_VEL
LIN {X 0,Y 62.275,Z 518.756,A -85,B 0,C 180,E1 -29000.645,E2 -29000.645} C_VEL
LIN {X 0,Y 65.204,Z 503.421,A -85,B 0,C 180,E1 -29009.506,E2 -29009.506} C_VEL
LIN {X 0,Y 68.415,Z 488.159,A -85,B 0,C 180,E1 -29016.198,E2 -29016.198} C_VEL
LIN {X 0,Y 71.762,Z 472.343,A -85,B 0,C 180,E1 -29021.375,E2 -29021.375} C_VEL
LIN {X 0,Y 74.915,Z 455.447,A -85,B 0,C 180,E1 -29025.423,E2 -29025.423} C_VEL
LIN {X 0,Y 80.284,Z 420.433,A -85,B 0,C 180,E1 -29031.486,E2 -29031.486} C_VEL
LIN {X 0,Y 80.61,Z 414.714,A -85,B 0,C 180,E1 -29032.531,E2 -29032.531} C_VEL
LIN {X 0,Y 78.37,Z 395.939,A -85,B 0,C 180,E1 -29036.917,E2 -29036.917} C_VEL
LIN {X 0,Y 78.829,Z 390.223,A -85,B 0,C 180,E1 -29037.948,E2 -29037.948} C_VEL
LIN {X 0,Y 79.89,Z 383.392,A -85,B 0,C 180,E1 -29039.008,E2 -29039.008} C_VEL
LIN {X 0,Y 71.857,Z 359.965,A -85,B 0,C 180,E1 -29047.518,E2 -29047.518} C_VEL
LIN {X 0,Y 66.83,Z 346.287,A -85,B 0,C 180,E1 -29053.967,E2 -29053.967} C_VEL
LIN {X 0,Y 62.661,Z 336.595,A -85,B 0,C 180,E1 -29059.963,E2 -29059.963} C_VEL
LIN {X 0,Y 59.241,Z 329.211,A -85,B 0,C 180,E1 -29065.739,E2 -29065.739} C_VEL
LIN {X 0,Y 56.918,Z 324.791,A -85,B 0,C 180,E1 -29070.209,E2 -29070.209} C_VEL
LIN {X 0,Y 55.544,Z 321.922,A -85,B 0,C 180,E1 -29073.254,E2 -29073.254} C_VEL
LIN {X 0,Y 52.747,Z 319.693,A -85,B 0,C 180,E1 -29078.852,E2 -29078.852} C_VEL
LIN {X 0,Y 51.668,Z 317.334,A -85,B 0,C 180,E1 -29082.26,E2 -29082.26} C_VEL
LIN {X 0,Y 51.566,Z 316.685,A -85,B 0,C 180,E1 -29083.035,E2 -29083.035} C_VEL
LIN {X 0,Y 51.385,Z 316.703,A -85,B 0,C 180,E1 -29086.808,E2 -29086.808} C_VEL
LIN {X 0,Y 51.014,Z 316.752,A -85,B 0,C 180,E1 -29094.4,E2 -29094.4} C_VEL
LIN {X 0,Y 50.995,Z 316.75,A -85,B 0,C 180,E1 -29104.23,E2 -29104.23} C_VEL
LIN {X 0,Y 50.968,Z 316.752,A -85,B 0,C 180,E1 -29113.571,E2 -29113.571} C_VEL
LIN {X 0,Y 51.016,Z 316.755,A -85,B 0,C 180,E1 -29125.727,E2 -29125.727} C_VEL
LIN {X 0,Y 51.012,Z 316.756,A -85,B 0,C 180,E1 -29135.594,E2 -29135.594} C_VEL
LIN {X 0,Y 51.539,Z 316.796,A -85,B 0,C 180,E1 -29144.94,E2 -29144.94} C_VEL
LIN {X 0,Y 52.708,Z 319.743,A -85,B 0,C 180,E1 -29148.956,E2 -29148.956} C_VEL
LIN {X 0,Y 55.147,Z 321.827,A -85,B 0,C 180,E1 -29153.937,E2 -29153.937} C_VEL
LIN {X 0,Y 57.702,Z 325.931,A -85,B 0,C 180,E1 -29159.089,E2 -29159.089} C_VEL
LIN {X 0,Y 61.328,Z 333.219,A -85,B 0,C 180,E1 -29165.554,E2 -29165.554} C_VEL
LIN {X 0,Y 65.758,Z 343.496,A -85,B 0,C 180,E1 -29172.347,E2 -29172.347} C_VEL
LIN {X 0,Y 70.538,Z 355.908,A -85,B 0,C 180,E1 -29178.651,E2 -29178.651} C_VEL
LIN {X 0,Y 72.831,Z 363.719,A -85,B 0,C 180,E1 -29181.73,E2 -29181.73} C_VEL
LIN {X 0,Y 79.012,Z 386.782,A -85,B 0,C 180,E1 -29189.293,E2 -29189.293} C_VEL
LIN {X 0,Y 80.66,Z 393.459,A -85,B 0,C 180,E1 -29191.181,E2 -29191.181} C_VEL
LIN {X 0,Y 68.972,Z 463.688,A -85,B 0,C 180,E1 -29203.459,E2 -29203.459} C_VEL
LIN {X 0,Y 66.153,Z 479.009,A -85,B 0,C 180,E1 -29207.488,E2 -29207.488} C_VEL
LIN {X 0,Y 63.116,Z 493.963,A -85,B 0,C 180,E1 -29212.8,E2 -29212.8} C_VEL
LIN {X 0,Y 59.967,Z 509.15,A -85,B 0,C 180,E1 -29220.137,E2 -29220.137} C_VEL
LIN {X 0,Y 57.746,Z 522.541,A -85,B 0,C 180,E1 -29228.596,E2 -29228.596} C_VEL
LIN {X 0,Y 56.67,Z 535.853,A -85,B 0,C 180,E1 -29239.293,E2 -29239.293} C_VEL
LIN {X 0,Y 57.345,Z 546.97,A -85,B 0,C 180,E1 -29250.01,E2 -29250.01} C_VEL
LIN {X 0,Y 59.189,Z 555.293,A -85,B 0,C 180,E1 -29259.243,E2 -29259.243} C_VEL
LIN {X 0,Y 59.767,Z 557.195,A -85,B 0,C 180,E1 -29261.56,E2 -29261.56} C_VEL
LIN {X 0,Y 60.09,Z 559.65,A -85,B 0,C 180,E1 -29265.651,E2 -29265.651} C_VEL
LIN {X 0,Y 62.17,Z 566.493,A -85,B 0,C 180,E1 -29280.587,E2 -29280.587} C_VEL
LIN {X 0,Y 69.32,Z 572.884,A -85,B 0,C 180,E1 -29295.221,E2 -29295.221} C_VEL
LIN {X 0,Y 68.685,Z 572.248,A -85,B 0,C 180,E1 -29296.843,E2 -29296.843} C_VEL
LIN {X 0,Y 60.343,Z 562.651,A -85,B 0,C 180,E1 -29310.325,E2 -29310.325} C_VEL
LIN {X 0,Y 56.74,Z 554.5,A -85,B 0,C 180,E1 -29321.956,E2 -29321.956} C_VEL
LIN {X 0,Y 55.046,Z 547.562,A -85,B 0,C 180,E1 -29330.811,E2 -29330.811} C_VEL
LIN {X 0,Y 54.054,Z 539.392,A -85,B 0,C 180,E1 -29339.994,E2 -29339.994} C_VEL
LIN {X 0,Y 54.318,Z 526.779,A -85,B 0,C 180,E1 -29352.131,E2 -29352.131} C_VEL
LIN {X 0,Y 55.958,Z 513.941,A -85,B 0,C 180,E1 -29362.128,E2 -29362.128} C_VEL
LIN {X 0,Y 59.037,Z 498.273,A -85,B 0,C 180,E1 -29371.552,E2 -29371.552} C_VEL
LIN {X 0,Y 62.74,Z 481.176,A -85,B 0,C 180,E1 -29379.048,E2 -29379.048} C_VEL
LIN {X 0,Y 66.135,Z 464.947,A -85,B 0,C 180,E1 -29384.21,E2 -29384.21} C_VEL
LIN {X 0,Y 69.243,Z 447.325,A -85,B 0,C 180,E1 -29388.184,E2 -29388.184} C_VEL
LIN {X 0,Y 78.829,Z 390.223,A -85,B 0,C 180,E1 -29397.948,E2 -29397.948} C_VEL
LIN {X 0,Y 78.682,Z 387.216,A -85,B 0,C 180,E1 -29398.616,E2 -29398.616} C_VEL
LIN {X 0,Y 76.82,Z 383.509,A -85,B 0,C 180,E1 -29400.026,E2 -29400.026} C_VEL
LIN {X 0,Y 70.507,Z 375.939,A -85,B 0,C 180,E1 -29404.29,E2 -29404.29} C_VEL
LIN {X 0,Y 69.464,Z 373.63,A -85,B 0,C 180,E1 -29405.325,E2 -29405.325} C_VEL
LIN {X 0,Y 64.503,Z 358.422,A -85,B 0,C 180,E1 -29412.07,E2 -29412.07} C_VEL
LIN {X 0,Y 60.289,Z 346.668,A -85,B 0,C 180,E1 -29418.702,E2 -29418.702} C_VEL
LIN {X 0,Y 55.88,Z 336.048,A -85,B 0,C 180,E1 -29426.836,E2 -29426.836} C_VEL
LIN {X 0,Y 52.859,Z 329.702,A -85,B 0,C 180,E1 -29433.563,E2 -29433.563} C_VEL
LIN {X 0,Y 51.999,Z 327.938,A -85,B 0,C 180,E1 -29435.807,E2 -29435.807} C_VEL
LIN {X 0,Y 49.362,Z 325.19,A -85,B 0,C 180,E1 -29442.316,E2 -29442.316} C_VEL
LIN {X 0,Y 48.397,Z 323.093,A -85,B 0,C 180,E1 -29446.006,E2 -29446.006} C_VEL
LIN {X 0,Y 44.981,Z 320.621,A -85,B 0,C 180,E1 -29461.301,E2 -29461.301} C_VEL
LIN {X 0,Y 44.609,Z 320.011,A -85,B 0,C 180,E1 -29465.209,E2 -29465.209} C_VEL
LIN {X 0,Y 44.361,Z 319.382,A -85,B 0,C 180,E1 -29476.711,E2 -29476.711} C_VEL
LIN {X 0,Y 45.198,Z 320.934,A -85,B 0,C 180,E1 -29488.354,E2 -29488.354} C_VEL
LIN {X 0,Y 48.629,Z 323.447,A -85,B 0,C 180,E1 -29502.664,E2 -29502.664} C_VEL
LIN {X 0,Y 50.334,Z 326.643,A -85,B 0,C 180,E1 -29508.334,E2 -29508.334} C_VEL
LIN {X 0,Y 52.258,Z 328.447,A -85,B 0,C 180,E1 -29512.69,E2 -29512.69} C_VEL
LIN {X 0,Y 53.784,Z 331.274,A -85,B 0,C 180,E1 -29516.265,E2 -29516.265} C_VEL
LIN {X 0,Y 56.792,Z 337.781,A -85,B 0,C 180,E1 -29522.682,E2 -29522.682} C_VEL
LIN {X 0,Y 60.784,Z 347.808,A -85,B 0,C 180,E1 -29529.925,E2 -29529.925} C_VEL
LIN {X 0,Y 65.128,Z 359.822,A -85,B 0,C 180,E1 -29536.577,E2 -29536.577} C_VEL
LIN {X 0,Y 68.643,Z 373.159,A -85,B 0,C 180,E1 -29541.995,E2 -29541.995} C_VEL
LIN {X 0,Y 73.981,Z 394.111,A -85,B 0,C 180,E1 -29549.164,E2 -29549.164} C_VEL
LIN {X 0,Y 62.042,Z 463.029,A -85,B 0,C 180,E1 -29562.3,E2 -29562.3} C_VEL
LIN {X 0,Y 59.245,Z 477.796,A -85,B 0,C 180,E1 -29566.605,E2 -29566.605} C_VEL
LIN {X 0,Y 55.797,Z 494.327,A -85,B 0,C 180,E1 -29573.265,E2 -29573.265} C_VEL
LIN {X 0,Y 52.894,Z 508.646,A -85,B 0,C 180,E1 -29581.219,E2 -29581.219} C_VEL
LIN {X 0,Y 50.877,Z 521.854,A -85,B 0,C 180,E1 -29590.86,E2 -29590.86} C_VEL
LIN {X 0,Y 50.263,Z 534.057,A -85,B 0,C 180,E1 -29601.974,E2 -29601.974} C_VEL
LIN {X 0,Y 51.505,Z 545.209,A -85,B 0,C 180,E1 -29613.923,E2 -29613.923} C_VEL
LIN {X 0,Y 53.774,Z 552.931,A -85,B 0,C 180,E1 -29623.232,E2 -29623.232} C_VEL
LIN {X 0,Y 54.255,Z 554.282,A -85,B 0,C 180,E1 -29625.025,E2 -29625.025} C_VEL
LIN {X 0,Y 54.626,Z 556.661,A -85,B 0,C 180,E1 -29629.557,E2 -29629.557} C_VEL
LIN {X 0,Y 58.316,Z 564.061,A -85,B 0,C 180,E1 -29647.066,E2 -29647.066} C_VEL
LIN {X 0,Y 61.383,Z 566.755,A -85,B 0,C 180,E1 -29653.402,E2 -29653.402} C_VEL
LIN {X 0,Y 61.781,Z 566.931,A -85,B 0,C 180,E1 -29655.806,E2 -29655.806} C_VEL
LIN {X 0,Y 54.269,Z 557.983,A -85,B 0,C 180,E1 -29668.795,E2 -29668.795} C_VEL
LIN {X 0,Y 50.865,Z 550.61,A -85,B 0,C 180,E1 -29679.786,E2 -29679.786} C_VEL
LIN {X 0,Y 48.831,Z 543.244,A -85,B 0,C 180,E1 -29689.629,E2 -29689.629} C_VEL
LIN {X 0,Y 47.629,Z 534.553,A -85,B 0,C 180,E1 -29699.993,E2 -29699.993} C_VEL
LIN {X 0,Y 47.727,Z 524.474,A -85,B 0,C 180,E1 -29710.6,E2 -29710.6} C_VEL
LIN {X 0,Y 49.464,Z 510.02,A -85,B 0,C 180,E1 -29722.993,E2 -29722.993} C_VEL
LIN {X 0,Y 52.049,Z 497.107,A -85,B 0,C 180,E1 -29731.541,E2 -29731.541} C_VEL
